# B&R Automation Studio project AAU12Segmenter
Automation Studio 4.12.2.93; technology packages: mapp 5.16.1, mapp6D 1.2.47924, mappCockpit 5.16.0, mappMotion 5.16.2, mappView 5.16.1, mappVision 5.16.1

## Configuration Config1

CPU X20CP1685, AutomationRuntime B4.91, Build 6.3.0, Safety 0.0, Vc V4.72.3

### Task classes (Cpu.sw)
```
Cyclic#1 (cycle 1000 us, tolerance 0 us):
  Main <- Modules.Main.Main.prg
  Acopos6D <- Modules.Acopos6D.Acopos6D.prg
  Vision <- Modules.Services.HMI.Vision.Vision.prg
  Vi_main <- Modules.Services.HMI.Vision.Vi_main.prg
  CTRL <- Modules.KUKA.CTRL.prg
Cyclic#4:
  HMI <- Modules.Services.HMI.HMI.prg
NcDataObjects: mcdrivelog
Binaries: FWRules, arcoal, arsvcreg, TCData, arflatprv, udbdef, mvLoader, mCoWebSc, User, iomap, Config_1, Role, arconfig, asfw, ashwac, sysconf, ashwd, Config_2, viApp, viComp, Settings, Settings_1, asnxdb1
Libraries: standard, brdkMU, brdkSTR, AsSem, sys_lib, brsystem, runtime, AsBrStr, McBase, AsZip, FileIO, AsARCfg, AsEPL, AsIO, astime, ViBase, IecCheck, CoTrace, brdkViBase, brdkViCal, brdkViGeom, brdkViImg, brdkViMapp, brdkViVF, BRSE_RTK, AsHttp, powerlnk, MTLinAlg, McAcp6D, SfDomain, MpBase, KUKAmxA3_1, AsIecCon, MpSfDomMgr, SfDomDrv, SfDomVis, asiodiag, aruser, asusb, arssl, astcp, AsUDP, asstring
```

### Hardware
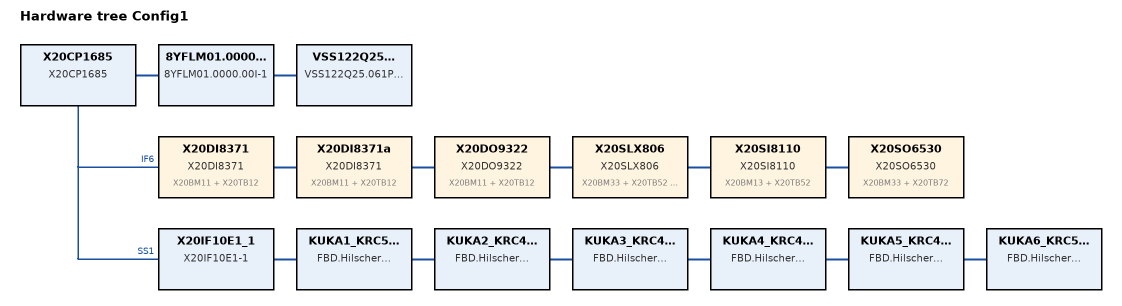
```
8YFLM01.0000.00I-1 : 8YFLM01.0000.00I-1 v0.0.0.1  [PLK1 -> X20CP1685.IF3 (NodeNumber=20) [Cable Type=PowerlinkCable, Length=10, Version=1.0.0.3]; PLK2 -> VSS122Q25.061P-000.PLK1 (NodeNumber=20) [Cable Type=PowerlinkCable, Length=10, Version=1.0.0.3]]
  Supervision = off
KUKA1_KRC5_ProfiNet_6_0 : FBD.Hilscher.PNIOGenDevDTM2.KUKA.PROFINET 6.0 v6.0 (OrderNumber=KUKA.PROFINET 6.0, VendorAddress=krc5-kuka1)  [PN1 -> X20IF10E1_1.IF1]
  DtmId = ed41ecf2-1ee6-4f16-8b0b-5a01acdc12f0
KUKA2_KRC4_ProfiNet_5_0 : FBD.Hilscher.PNIOGenDevDTM2.KRC4-ProfiNet_5.0 v5.0 (OrderNumber=KRC4-ProfiNet_5.0, VendorAddress=krc4-kuka2)  [PN1 -> KUKA1_KRC5_ProfiNet_6_0.PN2]
  DtmId = 37a7288f-95e5-4596-a95a-4f98395b86d6
KUKA3_KRC4_ProfiNet_5_0 : FBD.Hilscher.PNIOGenDevDTM2.KRC4-ProfiNet_5.0 v5.0 (OrderNumber=KRC4-ProfiNet_5.0, VendorAddress=krc4-kuka3)  [PN1 -> KUKA2_KRC4_ProfiNet_5_0.PN2]
  DtmId = 4619762a-1bda-4186-a1d7-16f7a0121dc3
KUKA4_KRC4_ProfiNet_5_0 : FBD.Hilscher.PNIOGenDevDTM2.KRC4-ProfiNet_5.0 v5.0 (OrderNumber=KRC4-ProfiNet_5.0, VendorAddress=krc4-kuka4)  [PN1 -> KUKA3_KRC4_ProfiNet_5_0.PN2]
  DtmId = 587b3b89-59c9-4dff-ae3f-6513934acbe2
KUKA5_KRC4_ProfiNet_5_0 : FBD.Hilscher.PNIOGenDevDTM2.KRC4-ProfiNet_5.0 v5.0 (OrderNumber=KRC4-ProfiNet_5.0, VendorAddress=krc4-kuka5)  [PN1 -> KUKA4_KRC4_ProfiNet_5_0.PN2]
  DtmId = 53f0387d-dc6f-4ff4-995c-9012f8d162e6
KUKA6_KRC5_ProfiNet_6_0 : FBD.Hilscher.PNIOGenDevDTM2.KUKA.PROFINET 6.0 v6.0 (OrderNumber=KUKA.PROFINET 6.0, VendorAddress=krc5-kuka6)  [PN1 -> KUKA5_KRC4_ProfiNet_5_0.PN2]
  DtmId = 2ed1eaca-6452-4986-be94-ac49d0fbd28d
VSS122Q25.061P-000 : VSS122Q25.061P-000 v1.6.0.546  [PLK1 -> 8YFLM01.0000.00I-1.PLK2 (NodeNumber=8) [Cable Type=PowerlinkCable, Length=10, Version=1.0.0.3]]
  Supervision = off
  VisionConfig = gCamera
X20BM11 : X20BM11 v1.1.0.0  [X2X1 -> X20CP1685.IF6]
X20BM11a : X20BM11 v1.1.0.0  [X2X1 -> X20BM11.X2X2]
X20BM11b : X20BM11 v1.1.0.0  [X2X1 -> X20BM11a.X2X2]
X20BM13 : X20BM13 v1.1.0.0  [X2X1 -> X20BM33.X2X2]
X20BM33 : X20BM33 v1.1.0.0  [X2X1 -> X20BM11b.X2X2]
X20BM33a : X20BM33 v1.1.0.0  [X2X1 -> X20BM13.X2X2]
X20CP1685 : X20CP1685 v1.4.0.0
  Connector IF2:
    ActivateDevice = 1
    Mode = Manual
    InternetAddress = 192.168.10.116
    SubnetMask = 255.255.255.0
    ActivateSnmp = 2
  Connector IF3:
    MtuSize = 1500
    DNAConfiguration = manual
    CycleTime = 1000
    InternetAddress = 192.168.200.240
    SubnetMask = 255.255.255.0
  ConfigurationID = Mapp6DDemoKit_Config1
  Simulation = 1
  PermanentPvSize = 6000
  RemanentGlobalPvSize = 40960
  VolatileGlobalPvSize = 200000
  TimerDeviceType = EPLX2X
  TimerDevice = X20CP1685.IF3
  Cyclic1Duration = 1000
  Cyclic1Tolerance = 0
  Cyclic2Duration = 8000
  Cyclic2Tolerance = 16000
  FileDevice1
  FileDeviceName1 = 6DData
  FileDevicePath1 = C:\
  FtpUser1
  FtpUsername1 = admin
  FtpUserPassword1 = jjEtgDO18IYHMAyC5LDIr++62vvoTF/vocBmfWTI62I=  // admin
  FtpUserSalt1 = E9oQkUbZ
  FTPAccessRight1 = 0
  FTPdevice1 = ALL
  ActivateOpcUa = 1
  OpcUaInformationModels_PV_Version = 1
X20DI8371 : X20DI8371 v1.4.0.0  [SS1 -> X20TB12.SS; SL -> X20BM11.SL1]
  Supervision = off
X20DI8371a : X20DI8371 v1.4.0.0  [SS1 -> X20TB12a.SS; SL -> X20BM11a.SL1]
X20DO9322 : X20DO9322 v1.5.0.0  [SS1 -> X20TB12b.SS; SL -> X20BM11b.SL1]
X20IF10E1_1 : X20IF10E1-1 v1.3.0.0  [SS -> X20CP1685.SS1]
  Connector IF1:
    DtmRef = FBDIF.Hilscher.PNIOControllerDTM2.NETX 100 RE/PNM
    DtmId = 9d996fcc-0d20-45c6-b313-689b61703394
  ConfigFile = X20IF10E1_1.dtm
  ConfigModule = asnxdb1
  CycleTime = 1000
X20SI8110 : X20SI8110 v2.4.0.0  [SS1 -> X20TB52b.SS; SL -> X20BM13.SL1]
X20SLX806 : X20SLX806 v2.4.1.1  [SS1 -> X20TB52.SS; SS2 -> X20TB52a.SS; SL -> X20BM33.SL1]
X20SO6530 : X20SO6530 v2.5.0.0  [SS1 -> X20TB72.SS; SL -> X20BM33a.SL1]
  SafeModuleID = 3
X20TB12 : X20TB12 v1.0.0.0
X20TB12a : X20TB12 v1.0.0.0
X20TB12b : X20TB12 v1.0.0.0
X20TB52 : X20TB52 v1.0.0.2
X20TB52a : X20TB52 v1.0.0.2
X20TB52b : X20TB52 v1.0.0.2
X20TB72 : X20TB72 v1.0.0.2
```

### IoMap.iom - X20CP1685/IoMap.iom
```iecst
VAR_CONFIG

	Cyclic#1.::FBin.Array[0] AT %IW."8YFLM01.0000.00I-1".EPL_FB_IN_0_I2007_S01;
	Cyclic#1.::FBin.Array[1] AT %IW."8YFLM01.0000.00I-1".EPL_FB_IN_1_I2007_S02;
	Cyclic#1.::FBin.Array[2] AT %IW."8YFLM01.0000.00I-1".EPL_FB_IN_2_I2007_S03;
	Cyclic#1.::FBin.Array[3] AT %IW."8YFLM01.0000.00I-1".EPL_FB_IN_3_I2007_S04;
	Cyclic#1.::FBin.Array[4] AT %IW."8YFLM01.0000.00I-1".EPL_FB_IN_4_I2007_S05;
	Cyclic#1.::FBin.Array[5] AT %IW."8YFLM01.0000.00I-1".EPL_FB_IN_5_I2007_S06;
	Cyclic#1.::FBin.Array[6] AT %IW."8YFLM01.0000.00I-1".EPL_FB_IN_6_I2007_S07;
	Cyclic#1.::FBin.Array[7] AT %IW."8YFLM01.0000.00I-1".EPL_FB_IN_7_I2007_S08;
	Cyclic#1.::FBin.Array[8] AT %IW."8YFLM01.0000.00I-1".EPL_FB_IN_8_I2007_S09;
	Cyclic#1.::FBin.Array[9] AT %IW."8YFLM01.0000.00I-1".EPL_FB_IN_9_I2007_S0A;
	Cyclic#1.::FBin.Array[10] AT %IW."8YFLM01.0000.00I-1".EPL_FB_IN_10_I2007_S0B;
	Cyclic#1.::FBin.Array[11] AT %IW."8YFLM01.0000.00I-1".EPL_FB_IN_11_I2007_S0C;
	Cyclic#1.::FBin.Array[12] AT %IW."8YFLM01.0000.00I-1".EPL_FB_IN_12_I2007_S0D;
	Cyclic#1.::FBin.Array[13] AT %IW."8YFLM01.0000.00I-1".EPL_FB_IN_13_I2007_S0E;
	Cyclic#1.::FBin.Array[14] AT %IW."8YFLM01.0000.00I-1".EPL_FB_IN_14_I2007_S0F;
	Cyclic#1.::FBin.Array[15] AT %IW."8YFLM01.0000.00I-1".EPL_FB_IN_15_I2007_S10;
	Cyclic#1.::FBin.Array[16] AT %IW."8YFLM01.0000.00I-1".EPL_FB_IN_16_I2007_S11;
	Cyclic#1.::FBin.Array[17] AT %IW."8YFLM01.0000.00I-1".EPL_FB_IN_17_I2007_S12;
	Cyclic#1.::FBin.Array[18] AT %IW."8YFLM01.0000.00I-1".EPL_FB_IN_18_I2007_S13;
	Cyclic#1.::FBin.Array[19] AT %IW."8YFLM01.0000.00I-1".EPL_FB_IN_19_I2007_S14;
	Cyclic#1.::FBin.Array[20] AT %IW."8YFLM01.0000.00I-1".EPL_FB_IN_20_I2007_S15;
	Cyclic#1.::FBin.Array[21] AT %IW."8YFLM01.0000.00I-1".EPL_FB_IN_21_I2007_S16;
	Cyclic#1.::FBin.Array[22] AT %IW."8YFLM01.0000.00I-1".EPL_FB_IN_22_I2007_S17;
	Cyclic#1.::FBin.Array[23] AT %IW."8YFLM01.0000.00I-1".EPL_FB_IN_23_I2007_S18;
	Cyclic#1.::FBin.Array[24] AT %IW."8YFLM01.0000.00I-1".EPL_FB_IN_24_I2007_S19;
	Cyclic#1.::FBin.Array[25] AT %IW."8YFLM01.0000.00I-1".EPL_FB_IN_25_I2007_S1A;
	Cyclic#1.::FBin.Array[26] AT %IW."8YFLM01.0000.00I-1".EPL_FB_IN_26_I2007_S1B;
	Cyclic#1.::FBin.Array[27] AT %IW."8YFLM01.0000.00I-1".EPL_FB_IN_27_I2007_S1C;
	Cyclic#1.::FBin.Array[28] AT %IW."8YFLM01.0000.00I-1".EPL_FB_IN_28_I2007_S1D;
	Cyclic#1.::FBin.Array[29] AT %IW."8YFLM01.0000.00I-1".EPL_FB_IN_29_I2007_S1E;
	Cyclic#1.::FBin.Array[30] AT %IW."8YFLM01.0000.00I-1".EPL_FB_IN_30_I2007_S1F;
	Cyclic#1.::FBin.Array[31] AT %IW."8YFLM01.0000.00I-1".EPL_FB_IN_31_I2007_S20;
	Cyclic#1.::FBin.Array[32] AT %IW."8YFLM01.0000.00I-1".EPL_FB_IN_32_I2007_S21;
	Cyclic#1.::FBin.Array[33] AT %IW."8YFLM01.0000.00I-1".EPL_FB_IN_33_I2007_S22;
	Cyclic#1.::FBin.Array[34] AT %IW."8YFLM01.0000.00I-1".EPL_FB_IN_34_I2007_S23;
	Cyclic#1.::FBin.Array[35] AT %IW."8YFLM01.0000.00I-1".EPL_FB_IN_35_I2007_S24;
	Cyclic#1.::FBin.Array[36] AT %IW."8YFLM01.0000.00I-1".EPL_FB_IN_36_I2007_S25;
	Cyclic#1.::FBin.Array[37] AT %IW."8YFLM01.0000.00I-1".EPL_FB_IN_37_I2007_S26;
	Cyclic#1.::FBin.Array[38] AT %IW."8YFLM01.0000.00I-1".EPL_FB_IN_38_I2007_S27;
	Cyclic#1.::FBin.Array[39] AT %IW."8YFLM01.0000.00I-1".EPL_FB_IN_39_I2007_S28;
	Cyclic#1.::FBin.Array[40] AT %IW."8YFLM01.0000.00I-1".EPL_FB_IN_40_I2007_S29;
	Cyclic#1.::FBin.Array[41] AT %IW."8YFLM01.0000.00I-1".EPL_FB_IN_41_I2007_S2A;
	Cyclic#1.::FBin.Array[42] AT %IW."8YFLM01.0000.00I-1".EPL_FB_IN_42_I2007_S2B;
	Cyclic#1.::FBin.Array[43] AT %IW."8YFLM01.0000.00I-1".EPL_FB_IN_43_I2007_S2C;
	Cyclic#1.::FBin.Array[44] AT %IW."8YFLM01.0000.00I-1".EPL_FB_IN_44_I2007_S2D;
	Cyclic#1.::FBin.Array[45] AT %IW."8YFLM01.0000.00I-1".EPL_FB_IN_45_I2007_S2E;
	Cyclic#1.::FBin.Array[46] AT %IW."8YFLM01.0000.00I-1".EPL_FB_IN_46_I2007_S2F;
	Cyclic#1.::FBin.Array[47] AT %IW."8YFLM01.0000.00I-1".EPL_FB_IN_47_I2007_S30;
	Cyclic#1.::FBin.Array[48] AT %IW."8YFLM01.0000.00I-1".EPL_FB_IN_48_I2007_S31;
	Cyclic#1.::FBin.Array[49] AT %IW."8YFLM01.0000.00I-1".EPL_FB_IN_49_I2007_S32;
	Cyclic#1.::FBin.Array[50] AT %IW."8YFLM01.0000.00I-1".EPL_FB_IN_50_I2007_S33;
	Cyclic#1.::FBin.Array[51] AT %IW."8YFLM01.0000.00I-1".EPL_FB_IN_51_I2007_S34;
	Cyclic#1.::FBin.Array[52] AT %IW."8YFLM01.0000.00I-1".EPL_FB_IN_52_I2007_S35;
	Cyclic#1.::FBin.Array[53] AT %IW."8YFLM01.0000.00I-1".EPL_FB_IN_53_I2007_S36;
	Cyclic#1.::FBin.Array[54] AT %IW."8YFLM01.0000.00I-1".EPL_FB_IN_54_I2007_S37;
	Cyclic#1.::FBin.Array[55] AT %IW."8YFLM01.0000.00I-1".EPL_FB_IN_55_I2007_S38;
	Cyclic#1.::FBin.Array[56] AT %IW."8YFLM01.0000.00I-1".EPL_FB_IN_56_I2007_S39;
	Cyclic#1.::FBin.Array[57] AT %IW."8YFLM01.0000.00I-1".EPL_FB_IN_57_I2007_S3A;
	Cyclic#1.::FBin.Array[58] AT %IW."8YFLM01.0000.00I-1".EPL_FB_IN_58_I2007_S3B;
	Cyclic#1.::FBin.Array[59] AT %IW."8YFLM01.0000.00I-1".EPL_FB_IN_59_I2007_S3C;
	Cyclic#1.::FBin.Array[60] AT %IW."8YFLM01.0000.00I-1".EPL_FB_IN_60_I2007_S3D;
	Cyclic#1.::FBin.Array[61] AT %IW."8YFLM01.0000.00I-1".EPL_FB_IN_61_I2007_S3E;
	Cyclic#1.::FBin.Array[62] AT %IW."8YFLM01.0000.00I-1".EPL_FB_IN_62_I2007_S3F;
	Cyclic#1.::FBin.Array[63] AT %IW."8YFLM01.0000.00I-1".EPL_FB_IN_63_I2007_S40;
	Cyclic#1.::FBin.Array[64] AT %IW."8YFLM01.0000.00I-1".EPL_FB_IN_64_I2007_S41;
	Cyclic#1.::FBin.Array[65] AT %IW."8YFLM01.0000.00I-1".EPL_FB_IN_65_I2007_S42;
	Cyclic#1.::FBin.Array[66] AT %IW."8YFLM01.0000.00I-1".EPL_FB_IN_66_I2007_S43;
	Cyclic#1.::FBin.Array[67] AT %IW."8YFLM01.0000.00I-1".EPL_FB_IN_67_I2007_S44;
	Cyclic#1.::FBin.Array[68] AT %IW."8YFLM01.0000.00I-1".EPL_FB_IN_68_I2007_S45;
	Cyclic#1.::FBin.Array[69] AT %IW."8YFLM01.0000.00I-1".EPL_FB_IN_69_I2007_S46;
	Cyclic#1.::FBin.Array[70] AT %IW."8YFLM01.0000.00I-1".EPL_FB_IN_70_I2007_S47;
	Cyclic#1.::FBin.Array[71] AT %IW."8YFLM01.0000.00I-1".EPL_FB_IN_71_I2007_S48;
	Cyclic#1.::FBin.Array[72] AT %IW."8YFLM01.0000.00I-1".EPL_FB_IN_72_I2007_S49;
	Cyclic#1.::FBin.Array[73] AT %IW."8YFLM01.0000.00I-1".EPL_FB_IN_73_I2007_S4A;
	Cyclic#1.::FBin.Array[74] AT %IW."8YFLM01.0000.00I-1".EPL_FB_IN_74_I2007_S4B;
	Cyclic#1.::FBin.Array[75] AT %IW."8YFLM01.0000.00I-1".EPL_FB_IN_75_I2007_S4C;
	Cyclic#1.::FBin.Array[76] AT %IW."8YFLM01.0000.00I-1".EPL_FB_IN_76_I2007_S4D;
	Cyclic#1.::FBin.Array[77] AT %IW."8YFLM01.0000.00I-1".EPL_FB_IN_77_I2007_S4E;
	Cyclic#1.::FBin.Array[78] AT %IW."8YFLM01.0000.00I-1".EPL_FB_IN_78_I2007_S4F;
	Cyclic#1.::FBin.Array[79] AT %IW."8YFLM01.0000.00I-1".EPL_FB_IN_79_I2007_S50;
	Cyclic#1.::FBin.Array[80] AT %IW."8YFLM01.0000.00I-1".EPL_FB_IN_80_I2007_S51;
	Cyclic#1.::FBin.Array[81] AT %IW."8YFLM01.0000.00I-1".EPL_FB_IN_81_I2007_S52;
	Cyclic#1.::FBin.Array[82] AT %IW."8YFLM01.0000.00I-1".EPL_FB_IN_82_I2007_S53;
	Cyclic#1.::FBin.Array[83] AT %IW."8YFLM01.0000.00I-1".EPL_FB_IN_83_I2007_S54;
	Cyclic#1.::FBin.Array[84] AT %IW."8YFLM01.0000.00I-1".EPL_FB_IN_84_I2007_S55;
	Cyclic#1.::FBin.Array[85] AT %IW."8YFLM01.0000.00I-1".EPL_FB_IN_85_I2007_S56;
	Cyclic#1.::FBin.Array[86] AT %IW."8YFLM01.0000.00I-1".EPL_FB_IN_86_I2007_S57;
	Cyclic#1.::FBin.Array[87] AT %IW."8YFLM01.0000.00I-1".EPL_FB_IN_87_I2007_S58;
	Cyclic#1.::FBin.Array[88] AT %IW."8YFLM01.0000.00I-1".EPL_FB_IN_88_I2007_S59;
	Cyclic#1.::FBin.Array[89] AT %IW."8YFLM01.0000.00I-1".EPL_FB_IN_89_I2007_S5A;
	Cyclic#1.::FBin.Array[90] AT %IW."8YFLM01.0000.00I-1".EPL_FB_IN_90_I2007_S5B;
	Cyclic#1.::FBin.Array[91] AT %IW."8YFLM01.0000.00I-1".EPL_FB_IN_91_I2007_S5C;
	Cyclic#1.::FBin.Array[92] AT %IW."8YFLM01.0000.00I-1".EPL_FB_IN_92_I2007_S5D;
	Cyclic#1.::FBin.Array[93] AT %IW."8YFLM01.0000.00I-1".EPL_FB_IN_93_I2007_S5E;
	Cyclic#1.::FBin.Array[94] AT %IW."8YFLM01.0000.00I-1".EPL_FB_IN_94_I2007_S5F;
	Cyclic#1.::FBin.Array[95] AT %IW."8YFLM01.0000.00I-1".EPL_FB_IN_95_I2007_S60;
	Cyclic#1.::FBin.Array[96] AT %IW."8YFLM01.0000.00I-1".EPL_FB_IN_96_I2007_S61;
	Cyclic#1.::FBin.Array[97] AT %IW."8YFLM01.0000.00I-1".EPL_FB_IN_97_I2007_S62;
	Cyclic#1.::FBin.Array[98] AT %IW."8YFLM01.0000.00I-1".EPL_FB_IN_98_I2007_S63;
	Cyclic#1.::FBin.Array[99] AT %IW."8YFLM01.0000.00I-1".EPL_FB_IN_99_I2007_S64;
	Cyclic#1.::FBin.Array[100] AT %IW."8YFLM01.0000.00I-1".EPL_FB_IN_100_I2007_S65;
	Cyclic#1.::FBin.Array[101] AT %IW."8YFLM01.0000.00I-1".EPL_FB_IN_101_I2007_S66;
	Cyclic#1.::FBin.Array[102] AT %IW."8YFLM01.0000.00I-1".EPL_FB_IN_102_I2007_S67;
	Cyclic#1.::FBin.Array[103] AT %IW."8YFLM01.0000.00I-1".EPL_FB_IN_103_I2007_S68;
	Cyclic#1.::FBin.Array[104] AT %IW."8YFLM01.0000.00I-1".EPL_FB_IN_104_I2007_S69;
	Cyclic#1.::FBin.Array[105] AT %IW."8YFLM01.0000.00I-1".EPL_FB_IN_105_I2007_S6A;
	Cyclic#1.::FBin.Array[106] AT %IW."8YFLM01.0000.00I-1".EPL_FB_IN_106_I2007_S6B;
	Cyclic#1.::FBin.Array[107] AT %IW."8YFLM01.0000.00I-1".EPL_FB_IN_107_I2007_S6C;
	Cyclic#1.::FBin.Array[108] AT %IW."8YFLM01.0000.00I-1".EPL_FB_IN_108_I2007_S6D;
	Cyclic#1.::FBin.Array[109] AT %IW."8YFLM01.0000.00I-1".EPL_FB_IN_109_I2007_S6E;
	Cyclic#1.::FBin.Array[110] AT %IW."8YFLM01.0000.00I-1".EPL_FB_IN_110_I2007_S6F;
	Cyclic#1.::FBin.Array[111] AT %IW."8YFLM01.0000.00I-1".EPL_FB_IN_111_I2007_S70;
	Cyclic#1.::FBin.Array[112] AT %IW."8YFLM01.0000.00I-1".EPL_FB_IN_112_I2007_S71;
	Cyclic#1.::FBin.Array[113] AT %IW."8YFLM01.0000.00I-1".EPL_FB_IN_113_I2007_S72;
	Cyclic#1.::FBin.Array[114] AT %IW."8YFLM01.0000.00I-1".EPL_FB_IN_114_I2007_S73;
	Cyclic#1.::FBin.Array[115] AT %IW."8YFLM01.0000.00I-1".EPL_FB_IN_115_I2007_S74;
	Cyclic#1.::FBin.Array[116] AT %IW."8YFLM01.0000.00I-1".EPL_FB_IN_116_I2007_S75;
	Cyclic#1.::FBin.Array[117] AT %IW."8YFLM01.0000.00I-1".EPL_FB_IN_117_I2007_S76;
	Cyclic#1.::FBin.Array[118] AT %IW."8YFLM01.0000.00I-1".EPL_FB_IN_118_I2007_S77;
	Cyclic#1.::FBin.Array[119] AT %IW."8YFLM01.0000.00I-1".EPL_FB_IN_119_I2007_S78;
	Cyclic#1.::FBin.Array[120] AT %IW."8YFLM01.0000.00I-1".EPL_FB_IN_120_I2007_S79;
	Cyclic#1.::FBin.Array[121] AT %IW."8YFLM01.0000.00I-1".EPL_FB_IN_121_I2007_S7A;
	Cyclic#1.::FBin.Array[122] AT %IW."8YFLM01.0000.00I-1".EPL_FB_IN_122_I2007_S7B;
	Cyclic#1.::FBin.Array[123] AT %IW."8YFLM01.0000.00I-1".EPL_FB_IN_123_I2007_S7C;
	Cyclic#1.::FBin.Array[124] AT %IW."8YFLM01.0000.00I-1".EPL_FB_IN_124_I2007_S7D;
	Cyclic#1.::FBin.Array[125] AT %IW."8YFLM01.0000.00I-1".EPL_FB_IN_125_I2007_S7E;
	Cyclic#1.::FBin.Array[126] AT %IW."8YFLM01.0000.00I-1".EPL_FB_IN_126_I2007_S7F;
	Cyclic#1.::FBin.Array[127] AT %IW."8YFLM01.0000.00I-1".EPL_FB_IN_127_I2007_S80;
	Cyclic#1.::FBin.Array[128] AT %IW."8YFLM01.0000.00I-1".EPL_FB_IN_128_I2007_S81;
	Cyclic#1.::FBin.Array[129] AT %IW."8YFLM01.0000.00I-1".EPL_FB_IN_129_I2007_S82;
	Cyclic#1.::FBin.Array[130] AT %IW."8YFLM01.0000.00I-1".EPL_FB_IN_130_I2007_S83;
	Cyclic#1.::FBin.Array[131] AT %IW."8YFLM01.0000.00I-1".EPL_FB_IN_131_I2007_S84;
	Cyclic#1.::FBin.Array[132] AT %IW."8YFLM01.0000.00I-1".EPL_FB_IN_132_I2007_S85;
	Cyclic#1.::FBin.Array[133] AT %IW."8YFLM01.0000.00I-1".EPL_FB_IN_133_I2007_S86;
	Cyclic#1.::FBin.Array[134] AT %IW."8YFLM01.0000.00I-1".EPL_FB_IN_134_I2007_S87;
	Cyclic#1.::FBin.Array[135] AT %IW."8YFLM01.0000.00I-1".EPL_FB_IN_135_I2007_S88;
	Cyclic#1.::FBin.Array[136] AT %IW."8YFLM01.0000.00I-1".EPL_FB_IN_136_I2007_S89;
	Cyclic#1.::FBin.Array[137] AT %IW."8YFLM01.0000.00I-1".EPL_FB_IN_137_I2007_S8A;
	Cyclic#1.::FBin.Array[138] AT %IW."8YFLM01.0000.00I-1".EPL_FB_IN_138_I2007_S8B;
	Cyclic#1.::FBin.Array[139] AT %IW."8YFLM01.0000.00I-1".EPL_FB_IN_139_I2007_S8C;
	Cyclic#1.::FBin.Array[140] AT %IW."8YFLM01.0000.00I-1".EPL_FB_IN_140_I2007_S8D;
	Cyclic#1.::FBin.Array[141] AT %IW."8YFLM01.0000.00I-1".EPL_FB_IN_141_I2007_S8E;
	Cyclic#1.::FBin.Array[142] AT %IW."8YFLM01.0000.00I-1".EPL_FB_IN_142_I2007_S8F;
	Cyclic#1.::FBin.Array[143] AT %IW."8YFLM01.0000.00I-1".EPL_FB_IN_143_I2007_S90;
	Cyclic#1.::FBin.Array[144] AT %IW."8YFLM01.0000.00I-1".EPL_FB_IN_144_I2007_S91;
	Cyclic#1.::FBin.Array[145] AT %IW."8YFLM01.0000.00I-1".EPL_FB_IN_145_I2007_S92;
	Cyclic#1.::FBin.Array[146] AT %IW."8YFLM01.0000.00I-1".EPL_FB_IN_146_I2007_S93;
	Cyclic#1.::FBin.Array[147] AT %IW."8YFLM01.0000.00I-1".EPL_FB_IN_147_I2007_S94;
	Cyclic#1.::FBin.Array[148] AT %IW."8YFLM01.0000.00I-1".EPL_FB_IN_148_I2007_S95;
	Cyclic#1.::FBin.Array[149] AT %IW."8YFLM01.0000.00I-1".EPL_FB_IN_149_I2007_S96;
	Cyclic#1.::FBin.Array[150] AT %IW."8YFLM01.0000.00I-1".EPL_FB_IN_150_I2007_S97;
	Cyclic#1.::FBin.Array[151] AT %IW."8YFLM01.0000.00I-1".EPL_FB_IN_151_I2007_S98;
	Cyclic#1.::FBin.Array[152] AT %IW."8YFLM01.0000.00I-1".EPL_FB_IN_152_I2007_S99;
	Cyclic#1.::FBin.Array[153] AT %IW."8YFLM01.0000.00I-1".EPL_FB_IN_153_I2007_S9A;
	Cyclic#1.::FBin.Array[154] AT %IW."8YFLM01.0000.00I-1".EPL_FB_IN_154_I2007_S9B;
	Cyclic#1.::FBin.Array[155] AT %IW."8YFLM01.0000.00I-1".EPL_FB_IN_155_I2007_S9C;
	Cyclic#1.::FBin.Array[156] AT %IW."8YFLM01.0000.00I-1".EPL_FB_IN_156_I2007_S9D;
	Cyclic#1.::FBin.Array[157] AT %IW."8YFLM01.0000.00I-1".EPL_FB_IN_157_I2007_S9E;
	Cyclic#1.::FBin.Array[158] AT %IW."8YFLM01.0000.00I-1".EPL_FB_IN_158_I2007_S9F;
	Cyclic#1.::FBin.Array[159] AT %IW."8YFLM01.0000.00I-1".EPL_FB_IN_159_I2007_SA0;
	Cyclic#1.::FBin.Array[160] AT %IW."8YFLM01.0000.00I-1".EPL_FB_IN_160_I2007_SA1;
	Cyclic#1.::FBin.Array[161] AT %IW."8YFLM01.0000.00I-1".EPL_FB_IN_161_I2007_SA2;
	Cyclic#1.::FBin.Array[162] AT %IW."8YFLM01.0000.00I-1".EPL_FB_IN_162_I2007_SA3;
	Cyclic#1.::FBin.Array[163] AT %IW."8YFLM01.0000.00I-1".EPL_FB_IN_163_I2007_SA4;
	Cyclic#1.::FBin.Array[164] AT %IW."8YFLM01.0000.00I-1".EPL_FB_IN_164_I2007_SA5;
	Cyclic#1.::FBin.Array[165] AT %IW."8YFLM01.0000.00I-1".EPL_FB_IN_165_I2007_SA6;
	Cyclic#1.::FBin.Array[166] AT %IW."8YFLM01.0000.00I-1".EPL_FB_IN_166_I2007_SA7;
	Cyclic#1.::FBin.Array[167] AT %IW."8YFLM01.0000.00I-1".EPL_FB_IN_167_I2007_SA8;
	Cyclic#1.::FBin.Array[168] AT %IW."8YFLM01.0000.00I-1".EPL_FB_IN_168_I2007_SA9;
	Cyclic#1.::FBin.Array[169] AT %IW."8YFLM01.0000.00I-1".EPL_FB_IN_169_I2007_SAA;
	Cyclic#1.::FBin.Array[170] AT %IW."8YFLM01.0000.00I-1".EPL_FB_IN_170_I2007_SAB;
	Cyclic#1.::FBin.Array[171] AT %IW."8YFLM01.0000.00I-1".EPL_FB_IN_171_I2007_SAC;
	Cyclic#1.::FBin.Array[172] AT %IW."8YFLM01.0000.00I-1".EPL_FB_IN_172_I2007_SAD;
	Cyclic#1.::FBin.Array[173] AT %IW."8YFLM01.0000.00I-1".EPL_FB_IN_173_I2007_SAE;
	Cyclic#1.::FBin.Array[174] AT %IW."8YFLM01.0000.00I-1".EPL_FB_IN_174_I2007_SAF;
	Cyclic#1.::FBin.Array[175] AT %IW."8YFLM01.0000.00I-1".EPL_FB_IN_175_I2007_SB0;
	Cyclic#1.::FBin.Array[176] AT %IW."8YFLM01.0000.00I-1".EPL_FB_IN_176_I2007_SB1;
	Cyclic#1.::FBin.Array[177] AT %IW."8YFLM01.0000.00I-1".EPL_FB_IN_177_I2007_SB2;
	Cyclic#1.::FBin.Array[178] AT %IW."8YFLM01.0000.00I-1".EPL_FB_IN_178_I2007_SB3;
	Cyclic#1.::FBin.Array[179] AT %IW."8YFLM01.0000.00I-1".EPL_FB_IN_179_I2007_SB4;
	Cyclic#1.::FBin.Array[180] AT %IW."8YFLM01.0000.00I-1".EPL_FB_IN_180_I2007_SB5;
	Cyclic#1.::FBin.Array[181] AT %IW."8YFLM01.0000.00I-1".EPL_FB_IN_181_I2007_SB6;
	Cyclic#1.::FBin.Array[182] AT %IW."8YFLM01.0000.00I-1".EPL_FB_IN_182_I2007_SB7;
	Cyclic#1.::FBin.Array[183] AT %IW."8YFLM01.0000.00I-1".EPL_FB_IN_183_I2007_SB8;
	Cyclic#1.::FBin.Array[184] AT %IW."8YFLM01.0000.00I-1".EPL_FB_IN_184_I2007_SB9;
	Cyclic#1.::FBin.Array[185] AT %IW."8YFLM01.0000.00I-1".EPL_FB_IN_185_I2007_SBA;
	Cyclic#1.::FBin.Array[186] AT %IW."8YFLM01.0000.00I-1".EPL_FB_IN_186_I2007_SBB;
	Cyclic#1.::FBin.Array[187] AT %IW."8YFLM01.0000.00I-1".EPL_FB_IN_187_I2007_SBC;
	Cyclic#1.::FBin.Array[188] AT %IW."8YFLM01.0000.00I-1".EPL_FB_IN_188_I2007_SBD;
	Cyclic#1.::FBin.Array[189] AT %IW."8YFLM01.0000.00I-1".EPL_FB_IN_189_I2007_SBE;
	Cyclic#1.::FBin.Array[190] AT %IW."8YFLM01.0000.00I-1".EPL_FB_IN_190_I2007_SBF;
	Cyclic#1.::FBin.Array[191] AT %IW."8YFLM01.0000.00I-1".EPL_FB_IN_191_I2007_SC0;
	Cyclic#1.::FBin.Array[192] AT %IW."8YFLM01.0000.00I-1".EPL_FB_IN_192_I2007_SC1;
	Cyclic#1.::FBin.Array[193] AT %IW."8YFLM01.0000.00I-1".EPL_FB_IN_193_I2007_SC2;
	Cyclic#1.::FBin.Array[194] AT %IW."8YFLM01.0000.00I-1".EPL_FB_IN_194_I2007_SC3;
	Cyclic#1.::FBin.Array[195] AT %IW."8YFLM01.0000.00I-1".EPL_FB_IN_195_I2007_SC4;
	Cyclic#1.::FBin.Array[196] AT %IW."8YFLM01.0000.00I-1".EPL_FB_IN_196_I2007_SC5;
	Cyclic#1.::FBin.Array[197] AT %IW."8YFLM01.0000.00I-1".EPL_FB_IN_197_I2007_SC6;
	Cyclic#1.::FBin.Array[198] AT %IW."8YFLM01.0000.00I-1".EPL_FB_IN_198_I2007_SC7;
	Cyclic#1.::FBin.Array[199] AT %IW."8YFLM01.0000.00I-1".EPL_FB_IN_199_I2007_SC8;
	Cyclic#1.::FBout.Array[0] AT %QW."8YFLM01.0000.00I-1".EPL_FB_OUT_0_I2008_S01Out;
	Cyclic#1.::FBout.Array[1] AT %QW."8YFLM01.0000.00I-1".EPL_FB_OUT_1_I2008_S02Out;
	Cyclic#1.::FBout.Array[2] AT %QW."8YFLM01.0000.00I-1".EPL_FB_OUT_2_I2008_S03Out;
	Cyclic#1.::FBout.Array[3] AT %QW."8YFLM01.0000.00I-1".EPL_FB_OUT_3_I2008_S04Out;
	Cyclic#1.::FBout.Array[4] AT %QW."8YFLM01.0000.00I-1".EPL_FB_OUT_4_I2008_S05Out;
	Cyclic#1.::FBout.Array[5] AT %QW."8YFLM01.0000.00I-1".EPL_FB_OUT_5_I2008_S06Out;
	Cyclic#1.::FBout.Array[6] AT %QW."8YFLM01.0000.00I-1".EPL_FB_OUT_6_I2008_S07Out;
	Cyclic#1.::FBout.Array[7] AT %QW."8YFLM01.0000.00I-1".EPL_FB_OUT_7_I2008_S08Out;
	Cyclic#1.::FBout.Array[8] AT %QW."8YFLM01.0000.00I-1".EPL_FB_OUT_8_I2008_S09Out;
	Cyclic#1.::FBout.Array[9] AT %QW."8YFLM01.0000.00I-1".EPL_FB_OUT_9_I2008_S0AOut;
	Cyclic#1.::FBout.Array[10] AT %QW."8YFLM01.0000.00I-1".EPL_FB_OUT_10_I2008_S0BOut;
	Cyclic#1.::FBout.Array[11] AT %QW."8YFLM01.0000.00I-1".EPL_FB_OUT_11_I2008_S0COut;
	Cyclic#1.::FBout.Array[12] AT %QW."8YFLM01.0000.00I-1".EPL_FB_OUT_12_I2008_S0DOut;
	Cyclic#1.::FBout.Array[13] AT %QW."8YFLM01.0000.00I-1".EPL_FB_OUT_13_I2008_S0EOut;
	Cyclic#1.::FBout.Array[14] AT %QW."8YFLM01.0000.00I-1".EPL_FB_OUT_14_I2008_S0FOut;
	Cyclic#1.::FBout.Array[15] AT %QW."8YFLM01.0000.00I-1".EPL_FB_OUT_15_I2008_S10Out;
	Cyclic#1.::FBout.Array[16] AT %QW."8YFLM01.0000.00I-1".EPL_FB_OUT_16_I2008_S11Out;
	Cyclic#1.::FBout.Array[17] AT %QW."8YFLM01.0000.00I-1".EPL_FB_OUT_17_I2008_S12Out;
	Cyclic#1.::FBout.Array[18] AT %QW."8YFLM01.0000.00I-1".EPL_FB_OUT_18_I2008_S13Out;
	Cyclic#1.::FBout.Array[19] AT %QW."8YFLM01.0000.00I-1".EPL_FB_OUT_19_I2008_S14Out;
	Cyclic#1.::FBout.Array[20] AT %QW."8YFLM01.0000.00I-1".EPL_FB_OUT_20_I2008_S15Out;
	Cyclic#1.::FBout.Array[21] AT %QW."8YFLM01.0000.00I-1".EPL_FB_OUT_21_I2008_S16Out;
	Cyclic#1.::FBout.Array[22] AT %QW."8YFLM01.0000.00I-1".EPL_FB_OUT_22_I2008_S17Out;
	Cyclic#1.::FBout.Array[23] AT %QW."8YFLM01.0000.00I-1".EPL_FB_OUT_23_I2008_S18Out;
	Cyclic#1.::FBout.Array[24] AT %QW."8YFLM01.0000.00I-1".EPL_FB_OUT_24_I2008_S19Out;
	Cyclic#1.::FBout.Array[25] AT %QW."8YFLM01.0000.00I-1".EPL_FB_OUT_25_I2008_S1AOut;
	Cyclic#1.::FBout.Array[26] AT %QW."8YFLM01.0000.00I-1".EPL_FB_OUT_26_I2008_S1BOut;
	Cyclic#1.::FBout.Array[27] AT %QW."8YFLM01.0000.00I-1".EPL_FB_OUT_27_I2008_S1COut;
	Cyclic#1.::FBout.Array[28] AT %QW."8YFLM01.0000.00I-1".EPL_FB_OUT_28_I2008_S1DOut;
	Cyclic#1.::FBout.Array[29] AT %QW."8YFLM01.0000.00I-1".EPL_FB_OUT_29_I2008_S1EOut;
	Cyclic#1.::FBout.Array[30] AT %QW."8YFLM01.0000.00I-1".EPL_FB_OUT_30_I2008_S1FOut;
	Cyclic#1.::FBout.Array[31] AT %QW."8YFLM01.0000.00I-1".EPL_FB_OUT_31_I2008_S20Out;
	Cyclic#1.::FBout.Array[32] AT %QW."8YFLM01.0000.00I-1".EPL_FB_OUT_32_I2008_S21Out;
	Cyclic#1.::FBout.Array[33] AT %QW."8YFLM01.0000.00I-1".EPL_FB_OUT_33_I2008_S22Out;
	Cyclic#1.::FBout.Array[34] AT %QW."8YFLM01.0000.00I-1".EPL_FB_OUT_34_I2008_S23Out;
	Cyclic#1.::FBout.Array[35] AT %QW."8YFLM01.0000.00I-1".EPL_FB_OUT_35_I2008_S24Out;
	Cyclic#1.::FBout.Array[36] AT %QW."8YFLM01.0000.00I-1".EPL_FB_OUT_36_I2008_S25Out;
	Cyclic#1.::FBout.Array[37] AT %QW."8YFLM01.0000.00I-1".EPL_FB_OUT_37_I2008_S26Out;
	Cyclic#1.::FBout.Array[38] AT %QW."8YFLM01.0000.00I-1".EPL_FB_OUT_38_I2008_S27Out;
	Cyclic#1.::FBout.Array[39] AT %QW."8YFLM01.0000.00I-1".EPL_FB_OUT_39_I2008_S28Out;
	Cyclic#1.::FBout.Array[40] AT %QW."8YFLM01.0000.00I-1".EPL_FB_OUT_40_I2008_S29Out;
	Cyclic#1.::FBout.Array[41] AT %QW."8YFLM01.0000.00I-1".EPL_FB_OUT_41_I2008_S2AOut;
	Cyclic#1.::FBout.Array[42] AT %QW."8YFLM01.0000.00I-1".EPL_FB_OUT_42_I2008_S2BOut;
	Cyclic#1.::FBout.Array[43] AT %QW."8YFLM01.0000.00I-1".EPL_FB_OUT_43_I2008_S2COut;
	Cyclic#1.::FBout.Array[44] AT %QW."8YFLM01.0000.00I-1".EPL_FB_OUT_44_I2008_S2DOut;
	Cyclic#1.::FBout.Array[45] AT %QW."8YFLM01.0000.00I-1".EPL_FB_OUT_45_I2008_S2EOut;
	Cyclic#1.::FBout.Array[46] AT %QW."8YFLM01.0000.00I-1".EPL_FB_OUT_46_I2008_S2FOut;
	Cyclic#1.::FBout.Array[47] AT %QW."8YFLM01.0000.00I-1".EPL_FB_OUT_47_I2008_S30Out;
	Cyclic#1.::FBout.Array[48] AT %QW."8YFLM01.0000.00I-1".EPL_FB_OUT_48_I2008_S31Out;
	Cyclic#1.::FBout.Array[49] AT %QW."8YFLM01.0000.00I-1".EPL_FB_OUT_49_I2008_S32Out;
	Cyclic#1.::FBout.Array[50] AT %QW."8YFLM01.0000.00I-1".EPL_FB_OUT_50_I2008_S33Out;
	Cyclic#1.::FBout.Array[51] AT %QW."8YFLM01.0000.00I-1".EPL_FB_OUT_51_I2008_S34Out;
	Cyclic#1.::FBout.Array[52] AT %QW."8YFLM01.0000.00I-1".EPL_FB_OUT_52_I2008_S35Out;
	Cyclic#1.::FBout.Array[53] AT %QW."8YFLM01.0000.00I-1".EPL_FB_OUT_53_I2008_S36Out;
	Cyclic#1.::FBout.Array[54] AT %QW."8YFLM01.0000.00I-1".EPL_FB_OUT_54_I2008_S37Out;
	Cyclic#1.::FBout.Array[55] AT %QW."8YFLM01.0000.00I-1".EPL_FB_OUT_55_I2008_S38Out;
	Cyclic#1.::FBout.Array[56] AT %QW."8YFLM01.0000.00I-1".EPL_FB_OUT_56_I2008_S39Out;
	Cyclic#1.::FBout.Array[57] AT %QW."8YFLM01.0000.00I-1".EPL_FB_OUT_57_I2008_S3AOut;
	Cyclic#1.::FBout.Array[58] AT %QW."8YFLM01.0000.00I-1".EPL_FB_OUT_58_I2008_S3BOut;
	Cyclic#1.::FBout.Array[59] AT %QW."8YFLM01.0000.00I-1".EPL_FB_OUT_59_I2008_S3COut;
	Cyclic#1.::FBout.Array[60] AT %QW."8YFLM01.0000.00I-1".EPL_FB_OUT_60_I2008_S3DOut;
	Cyclic#1.::FBout.Array[61] AT %QW."8YFLM01.0000.00I-1".EPL_FB_OUT_61_I2008_S3EOut;
	Cyclic#1.::FBout.Array[62] AT %QW."8YFLM01.0000.00I-1".EPL_FB_OUT_62_I2008_S3FOut;
	Cyclic#1.::FBout.Array[63] AT %QW."8YFLM01.0000.00I-1".EPL_FB_OUT_63_I2008_S40Out;
	Cyclic#1.::FBout.Array[64] AT %QW."8YFLM01.0000.00I-1".EPL_FB_OUT_64_I2008_S41Out;
	Cyclic#1.::FBout.Array[65] AT %QW."8YFLM01.0000.00I-1".EPL_FB_OUT_65_I2008_S42Out;
	Cyclic#1.::FBout.Array[66] AT %QW."8YFLM01.0000.00I-1".EPL_FB_OUT_66_I2008_S43Out;
	Cyclic#1.::FBout.Array[67] AT %QW."8YFLM01.0000.00I-1".EPL_FB_OUT_67_I2008_S44Out;
	Cyclic#1.::FBout.Array[68] AT %QW."8YFLM01.0000.00I-1".EPL_FB_OUT_68_I2008_S45Out;
	Cyclic#1.::FBout.Array[69] AT %QW."8YFLM01.0000.00I-1".EPL_FB_OUT_69_I2008_S46Out;
	Cyclic#1.::FBout.Array[70] AT %QW."8YFLM01.0000.00I-1".EPL_FB_OUT_70_I2008_S47Out;
	Cyclic#1.::FBout.Array[71] AT %QW."8YFLM01.0000.00I-1".EPL_FB_OUT_71_I2008_S48Out;
	Cyclic#1.::FBout.Array[72] AT %QW."8YFLM01.0000.00I-1".EPL_FB_OUT_72_I2008_S49Out;
	Cyclic#1.::FBout.Array[73] AT %QW."8YFLM01.0000.00I-1".EPL_FB_OUT_73_I2008_S4AOut;
	Cyclic#1.::FBout.Array[74] AT %QW."8YFLM01.0000.00I-1".EPL_FB_OUT_74_I2008_S4BOut;
	Cyclic#1.::FBout.Array[75] AT %QW."8YFLM01.0000.00I-1".EPL_FB_OUT_75_I2008_S4COut;
	Cyclic#1.::FBout.Array[76] AT %QW."8YFLM01.0000.00I-1".EPL_FB_OUT_76_I2008_S4DOut;
	Cyclic#1.::FBout.Array[77] AT %QW."8YFLM01.0000.00I-1".EPL_FB_OUT_77_I2008_S4EOut;
	Cyclic#1.::FBout.Array[78] AT %QW."8YFLM01.0000.00I-1".EPL_FB_OUT_78_I2008_S4FOut;
	Cyclic#1.::FBout.Array[79] AT %QW."8YFLM01.0000.00I-1".EPL_FB_OUT_79_I2008_S50Out;
	Cyclic#1.::FBout.Array[80] AT %QW."8YFLM01.0000.00I-1".EPL_FB_OUT_80_I2008_S51Out;
	Cyclic#1.::FBout.Array[81] AT %QW."8YFLM01.0000.00I-1".EPL_FB_OUT_81_I2008_S52Out;
	Cyclic#1.::FBout.Array[82] AT %QW."8YFLM01.0000.00I-1".EPL_FB_OUT_82_I2008_S53Out;
	Cyclic#1.::FBout.Array[83] AT %QW."8YFLM01.0000.00I-1".EPL_FB_OUT_83_I2008_S54Out;
	Cyclic#1.::FBout.Array[84] AT %QW."8YFLM01.0000.00I-1".EPL_FB_OUT_84_I2008_S55Out;
	Cyclic#1.::FBout.Array[85] AT %QW."8YFLM01.0000.00I-1".EPL_FB_OUT_85_I2008_S56Out;
	Cyclic#1.::FBout.Array[86] AT %QW."8YFLM01.0000.00I-1".EPL_FB_OUT_86_I2008_S57Out;
	Cyclic#1.::FBout.Array[87] AT %QW."8YFLM01.0000.00I-1".EPL_FB_OUT_87_I2008_S58Out;
	Cyclic#1.::FBout.Array[88] AT %QW."8YFLM01.0000.00I-1".EPL_FB_OUT_88_I2008_S59Out;
	Cyclic#1.::FBout.Array[89] AT %QW."8YFLM01.0000.00I-1".EPL_FB_OUT_89_I2008_S5AOut;
	Cyclic#1.::FBout.Array[90] AT %QW."8YFLM01.0000.00I-1".EPL_FB_OUT_90_I2008_S5BOut;
	Cyclic#1.::FBout.Array[91] AT %QW."8YFLM01.0000.00I-1".EPL_FB_OUT_91_I2008_S5COut;
	Cyclic#1.::FBout.Array[92] AT %QW."8YFLM01.0000.00I-1".EPL_FB_OUT_92_I2008_S5DOut;
	Cyclic#1.::FBout.Array[93] AT %QW."8YFLM01.0000.00I-1".EPL_FB_OUT_93_I2008_S5EOut;
	Cyclic#1.::FBout.Array[94] AT %QW."8YFLM01.0000.00I-1".EPL_FB_OUT_94_I2008_S5FOut;
	Cyclic#1.::FBout.Array[95] AT %QW."8YFLM01.0000.00I-1".EPL_FB_OUT_95_I2008_S60Out;
	Cyclic#1.::FBout.Array[96] AT %QW."8YFLM01.0000.00I-1".EPL_FB_OUT_96_I2008_S61Out;
	Cyclic#1.::FBout.Array[97] AT %QW."8YFLM01.0000.00I-1".EPL_FB_OUT_97_I2008_S62Out;
	Cyclic#1.::FBout.Array[98] AT %QW."8YFLM01.0000.00I-1".EPL_FB_OUT_98_I2008_S63Out;
	Cyclic#1.::FBout.Array[99] AT %QW."8YFLM01.0000.00I-1".EPL_FB_OUT_99_I2008_S64Out;
	Cyclic#1.::FBout.Array[100] AT %QW."8YFLM01.0000.00I-1".EPL_FB_OUT_100_I2008_S65Out;
	Cyclic#1.::FBout.Array[101] AT %QW."8YFLM01.0000.00I-1".EPL_FB_OUT_101_I2008_S66Out;
	Cyclic#1.::FBout.Array[102] AT %QW."8YFLM01.0000.00I-1".EPL_FB_OUT_102_I2008_S67Out;
	Cyclic#1.::FBout.Array[103] AT %QW."8YFLM01.0000.00I-1".EPL_FB_OUT_103_I2008_S68Out;
	Cyclic#1.::FBout.Array[104] AT %QW."8YFLM01.0000.00I-1".EPL_FB_OUT_104_I2008_S69Out;
	Cyclic#1.::FBout.Array[105] AT %QW."8YFLM01.0000.00I-1".EPL_FB_OUT_105_I2008_S6AOut;
	Cyclic#1.::FBout.Array[106] AT %QW."8YFLM01.0000.00I-1".EPL_FB_OUT_106_I2008_S6BOut;
	Cyclic#1.::FBout.Array[107] AT %QW."8YFLM01.0000.00I-1".EPL_FB_OUT_107_I2008_S6COut;
	Cyclic#1.::FBout.Array[108] AT %QW."8YFLM01.0000.00I-1".EPL_FB_OUT_108_I2008_S6DOut;
	Cyclic#1.::FBout.Array[109] AT %QW."8YFLM01.0000.00I-1".EPL_FB_OUT_109_I2008_S6EOut;
	Cyclic#1.::FBout.Array[110] AT %QW."8YFLM01.0000.00I-1".EPL_FB_OUT_110_I2008_S6FOut;
	Cyclic#1.::FBout.Array[111] AT %QW."8YFLM01.0000.00I-1".EPL_FB_OUT_111_I2008_S70Out;
	Cyclic#1.::FBout.Array[112] AT %QW."8YFLM01.0000.00I-1".EPL_FB_OUT_112_I2008_S71Out;
	Cyclic#1.::FBout.Array[113] AT %QW."8YFLM01.0000.00I-1".EPL_FB_OUT_113_I2008_S72Out;
	Cyclic#1.::FBout.Array[114] AT %QW."8YFLM01.0000.00I-1".EPL_FB_OUT_114_I2008_S73Out;
	Cyclic#1.::FBout.Array[115] AT %QW."8YFLM01.0000.00I-1".EPL_FB_OUT_115_I2008_S74Out;
	Cyclic#1.::FBout.Array[116] AT %QW."8YFLM01.0000.00I-1".EPL_FB_OUT_116_I2008_S75Out;
	Cyclic#1.::FBout.Array[117] AT %QW."8YFLM01.0000.00I-1".EPL_FB_OUT_117_I2008_S76Out;
	Cyclic#1.::FBout.Array[118] AT %QW."8YFLM01.0000.00I-1".EPL_FB_OUT_118_I2008_S77Out;
	Cyclic#1.::FBout.Array[119] AT %QW."8YFLM01.0000.00I-1".EPL_FB_OUT_119_I2008_S78Out;
	Cyclic#1.::FBout.Array[120] AT %QW."8YFLM01.0000.00I-1".EPL_FB_OUT_120_I2008_S79Out;
	Cyclic#1.::FBout.Array[121] AT %QW."8YFLM01.0000.00I-1".EPL_FB_OUT_121_I2008_S7AOut;
	Cyclic#1.::FBout.Array[122] AT %QW."8YFLM01.0000.00I-1".EPL_FB_OUT_122_I2008_S7BOut;
	Cyclic#1.::FBout.Array[123] AT %QW."8YFLM01.0000.00I-1".EPL_FB_OUT_123_I2008_S7COut;
	Cyclic#1.::FBout.Array[124] AT %QW."8YFLM01.0000.00I-1".EPL_FB_OUT_124_I2008_S7DOut;
	Cyclic#1.::FBout.Array[125] AT %QW."8YFLM01.0000.00I-1".EPL_FB_OUT_125_I2008_S7EOut;
	Cyclic#1.::FBout.Array[126] AT %QW."8YFLM01.0000.00I-1".EPL_FB_OUT_126_I2008_S7FOut;
	Cyclic#1.::FBout.Array[127] AT %QW."8YFLM01.0000.00I-1".EPL_FB_OUT_127_I2008_S80Out;
	Cyclic#1.::FBout.Array[128] AT %QW."8YFLM01.0000.00I-1".EPL_FB_OUT_128_I2008_S81Out;
	Cyclic#1.::FBout.Array[129] AT %QW."8YFLM01.0000.00I-1".EPL_FB_OUT_129_I2008_S82Out;
	Cyclic#1.::FBout.Array[130] AT %QW."8YFLM01.0000.00I-1".EPL_FB_OUT_130_I2008_S83Out;
	Cyclic#1.::FBout.Array[131] AT %QW."8YFLM01.0000.00I-1".EPL_FB_OUT_131_I2008_S84Out;
	Cyclic#1.::FBout.Array[132] AT %QW."8YFLM01.0000.00I-1".EPL_FB_OUT_132_I2008_S85Out;
	Cyclic#1.::FBout.Array[133] AT %QW."8YFLM01.0000.00I-1".EPL_FB_OUT_133_I2008_S86Out;
	Cyclic#1.::FBout.Array[134] AT %QW."8YFLM01.0000.00I-1".EPL_FB_OUT_134_I2008_S87Out;
	Cyclic#1.::FBout.Array[135] AT %QW."8YFLM01.0000.00I-1".EPL_FB_OUT_135_I2008_S88Out;
	Cyclic#1.::FBout.Array[136] AT %QW."8YFLM01.0000.00I-1".EPL_FB_OUT_136_I2008_S89Out;
	Cyclic#1.::FBout.Array[137] AT %QW."8YFLM01.0000.00I-1".EPL_FB_OUT_137_I2008_S8AOut;
	Cyclic#1.::FBout.Array[138] AT %QW."8YFLM01.0000.00I-1".EPL_FB_OUT_138_I2008_S8BOut;
	Cyclic#1.::FBout.Array[139] AT %QW."8YFLM01.0000.00I-1".EPL_FB_OUT_139_I2008_S8COut;
	Cyclic#1.::FBout.Array[140] AT %QW."8YFLM01.0000.00I-1".EPL_FB_OUT_140_I2008_S8DOut;
	Cyclic#1.::FBout.Array[141] AT %QW."8YFLM01.0000.00I-1".EPL_FB_OUT_141_I2008_S8EOut;
	Cyclic#1.::FBout.Array[142] AT %QW."8YFLM01.0000.00I-1".EPL_FB_OUT_142_I2008_S8FOut;
	Cyclic#1.::FBout.Array[143] AT %QW."8YFLM01.0000.00I-1".EPL_FB_OUT_143_I2008_S90Out;
	Cyclic#1.::FBout.Array[144] AT %QW."8YFLM01.0000.00I-1".EPL_FB_OUT_144_I2008_S91Out;
	Cyclic#1.::FBout.Array[145] AT %QW."8YFLM01.0000.00I-1".EPL_FB_OUT_145_I2008_S92Out;
	Cyclic#1.::FBout.Array[146] AT %QW."8YFLM01.0000.00I-1".EPL_FB_OUT_146_I2008_S93Out;
	Cyclic#1.::FBout.Array[147] AT %QW."8YFLM01.0000.00I-1".EPL_FB_OUT_147_I2008_S94Out;
	Cyclic#1.::FBout.Array[148] AT %QW."8YFLM01.0000.00I-1".EPL_FB_OUT_148_I2008_S95Out;
	Cyclic#1.::FBout.Array[149] AT %QW."8YFLM01.0000.00I-1".EPL_FB_OUT_149_I2008_S96Out;
	Cyclic#1.::FBout.Array[150] AT %QW."8YFLM01.0000.00I-1".EPL_FB_OUT_150_I2008_S97Out;
	Cyclic#1.::FBout.Array[151] AT %QW."8YFLM01.0000.00I-1".EPL_FB_OUT_151_I2008_S98Out;
	Cyclic#1.::FBout.Array[152] AT %QW."8YFLM01.0000.00I-1".EPL_FB_OUT_152_I2008_S99Out;
	Cyclic#1.::FBout.Array[153] AT %QW."8YFLM01.0000.00I-1".EPL_FB_OUT_153_I2008_S9AOut;
	Cyclic#1.::FBout.Array[154] AT %QW."8YFLM01.0000.00I-1".EPL_FB_OUT_154_I2008_S9BOut;
	Cyclic#1.::FBout.Array[155] AT %QW."8YFLM01.0000.00I-1".EPL_FB_OUT_155_I2008_S9COut;
	Cyclic#1.::FBout.Array[156] AT %QW."8YFLM01.0000.00I-1".EPL_FB_OUT_156_I2008_S9DOut;
	Cyclic#1.::FBout.Array[157] AT %QW."8YFLM01.0000.00I-1".EPL_FB_OUT_157_I2008_S9EOut;
	Cyclic#1.::FBout.Array[158] AT %QW."8YFLM01.0000.00I-1".EPL_FB_OUT_158_I2008_S9FOut;
	Cyclic#1.::FBout.Array[159] AT %QW."8YFLM01.0000.00I-1".EPL_FB_OUT_159_I2008_SA0Out;
	Cyclic#1.::FBout.Array[160] AT %QW."8YFLM01.0000.00I-1".EPL_FB_OUT_160_I2008_SA1Out;
	Cyclic#1.::FBout.Array[161] AT %QW."8YFLM01.0000.00I-1".EPL_FB_OUT_161_I2008_SA2Out;
	Cyclic#1.::FBout.Array[162] AT %QW."8YFLM01.0000.00I-1".EPL_FB_OUT_162_I2008_SA3Out;
	Cyclic#1.::FBout.Array[163] AT %QW."8YFLM01.0000.00I-1".EPL_FB_OUT_163_I2008_SA4Out;
	Cyclic#1.::FBout.Array[164] AT %QW."8YFLM01.0000.00I-1".EPL_FB_OUT_164_I2008_SA5Out;
	Cyclic#1.::FBout.Array[165] AT %QW."8YFLM01.0000.00I-1".EPL_FB_OUT_165_I2008_SA6Out;
	Cyclic#1.::FBout.Array[166] AT %QW."8YFLM01.0000.00I-1".EPL_FB_OUT_166_I2008_SA7Out;
	Cyclic#1.::FBout.Array[167] AT %QW."8YFLM01.0000.00I-1".EPL_FB_OUT_167_I2008_SA8Out;
	Cyclic#1.::FBout.Array[168] AT %QW."8YFLM01.0000.00I-1".EPL_FB_OUT_168_I2008_SA9Out;
	Cyclic#1.::FBout.Array[169] AT %QW."8YFLM01.0000.00I-1".EPL_FB_OUT_169_I2008_SAAOut;
	Cyclic#1.::FBout.Array[170] AT %QW."8YFLM01.0000.00I-1".EPL_FB_OUT_170_I2008_SABOut;
	Cyclic#1.::FBout.Array[171] AT %QW."8YFLM01.0000.00I-1".EPL_FB_OUT_171_I2008_SACOut;
	Cyclic#1.::FBout.Array[172] AT %QW."8YFLM01.0000.00I-1".EPL_FB_OUT_172_I2008_SADOut;
	Cyclic#1.::FBout.Array[173] AT %QW."8YFLM01.0000.00I-1".EPL_FB_OUT_173_I2008_SAEOut;
	Cyclic#1.::FBout.Array[174] AT %QW."8YFLM01.0000.00I-1".EPL_FB_OUT_174_I2008_SAFOut;
	Cyclic#1.::FBout.Array[175] AT %QW."8YFLM01.0000.00I-1".EPL_FB_OUT_175_I2008_SB0Out;
	Cyclic#1.::FBout.Array[176] AT %QW."8YFLM01.0000.00I-1".EPL_FB_OUT_176_I2008_SB1Out;
	Cyclic#1.::FBout.Array[177] AT %QW."8YFLM01.0000.00I-1".EPL_FB_OUT_177_I2008_SB2Out;
	Cyclic#1.::FBout.Array[178] AT %QW."8YFLM01.0000.00I-1".EPL_FB_OUT_178_I2008_SB3Out;
	Cyclic#1.::FBout.Array[179] AT %QW."8YFLM01.0000.00I-1".EPL_FB_OUT_179_I2008_SB4Out;
	Cyclic#1.::FBout.Array[180] AT %QW."8YFLM01.0000.00I-1".EPL_FB_OUT_180_I2008_SB5Out;
	Cyclic#1.::FBout.Array[181] AT %QW."8YFLM01.0000.00I-1".EPL_FB_OUT_181_I2008_SB6Out;
	Cyclic#1.::FBout.Array[182] AT %QW."8YFLM01.0000.00I-1".EPL_FB_OUT_182_I2008_SB7Out;
	Cyclic#1.::FBout.Array[183] AT %QW."8YFLM01.0000.00I-1".EPL_FB_OUT_183_I2008_SB8Out;
	Cyclic#1.::FBout.Array[184] AT %QW."8YFLM01.0000.00I-1".EPL_FB_OUT_184_I2008_SB9Out;
	Cyclic#1.::FBout.Array[185] AT %QW."8YFLM01.0000.00I-1".EPL_FB_OUT_185_I2008_SBAOut;
	Cyclic#1.::FBout.Array[186] AT %QW."8YFLM01.0000.00I-1".EPL_FB_OUT_186_I2008_SBBOut;
	Cyclic#1.::FBout.Array[187] AT %QW."8YFLM01.0000.00I-1".EPL_FB_OUT_187_I2008_SBCOut;
	Cyclic#1.::FBout.Array[188] AT %QW."8YFLM01.0000.00I-1".EPL_FB_OUT_188_I2008_SBDOut;
	Cyclic#1.::FBout.Array[189] AT %QW."8YFLM01.0000.00I-1".EPL_FB_OUT_189_I2008_SBEOut;
	Cyclic#1.::FBout.Array[190] AT %QW."8YFLM01.0000.00I-1".EPL_FB_OUT_190_I2008_SBFOut;
	Cyclic#1.::FBout.Array[191] AT %QW."8YFLM01.0000.00I-1".EPL_FB_OUT_191_I2008_SC0Out;
	Cyclic#1.::FBout.Array[192] AT %QW."8YFLM01.0000.00I-1".EPL_FB_OUT_192_I2008_SC1Out;
	Cyclic#1.::FBout.Array[193] AT %QW."8YFLM01.0000.00I-1".EPL_FB_OUT_193_I2008_SC2Out;
	Cyclic#1.::FBout.Array[194] AT %QW."8YFLM01.0000.00I-1".EPL_FB_OUT_194_I2008_SC3Out;
	Cyclic#1.::FBout.Array[195] AT %QW."8YFLM01.0000.00I-1".EPL_FB_OUT_195_I2008_SC4Out;
	Cyclic#1.::FBout.Array[196] AT %QW."8YFLM01.0000.00I-1".EPL_FB_OUT_196_I2008_SC5Out;
	Cyclic#1.::FBout.Array[197] AT %QW."8YFLM01.0000.00I-1".EPL_FB_OUT_197_I2008_SC6Out;
	Cyclic#1.::FBout.Array[198] AT %QW."8YFLM01.0000.00I-1".EPL_FB_OUT_198_I2008_SC7Out;
	Cyclic#1.::FBout.Array[199] AT %QW."8YFLM01.0000.00I-1".EPL_FB_OUT_199_I2008_SC8Out;
	Cyclic#1.::gVisionSensor[3].HW.Connected AT %IX."VSS122Q25.061P-000".ModuleOk;
	Cyclic#1.::gVisionSensor[3].HW.SerialNumber AT %ID."VSS122Q25.061P-000".SerialNumber;
	Cyclic#1.::gVisionSensor[3].HW.ID AT %ID."VSS122Q25.061P-000".ModuleID;
	Cyclic#1.::gVisionSensor[3].HW.Variant AT %ID."VSS122Q25.061P-000".HardwareVariant;
	Cyclic#1.::gVisionSensor[3].HW.Firmware AT %ID."VSS122Q25.061P-000".FirmwareVersion;
	Cyclic#1.::gVisionSensor[3].DAT.Exposure AT %QD."VSS122Q25.061P-000".ExposureTime01;
	Cyclic#1.::gVisionSensor[3].DAT.FlashSegment AT %QB."VSS122Q25.061P-000".FlashSegment01;
	Cyclic#1.::gVisionSensor[3].DAT.AutoSetupExposure AT %ID."VSS122Q25.061P-000".ReadExposureTime;
	Cyclic#1.::gVisionSensor[3].DAT.Status AT %ID."VSS122Q25.061P-000".CameraStatus;
	Cyclic#1.::gVisionSensor[3].DAT.AutoSetupFocus AT %IW."VSS122Q25.061P-000".ReadFocus;
	Cyclic#1.::gVisionSensor[3].DAT.Focus AT %QW."VSS122Q25.061P-000".SetFocus;
	Cyclic#1.::gVisionSensor[3].DAT.Gain AT %QB."VSS122Q25.061P-000".GainLevel;
	Cyclic#1.::gVisionSensor[3].DAT.AutoSetupGain AT %IB."VSS122Q25.061P-000".ReadGainLevel;
	Cyclic#1.::gVisionSensor[3].DAT.AcquisitionFailedCnt AT %IB."VSS122Q25.061P-000".FailedAcquisitionCnt;
	Cyclic#1.::gVisionSensor[3].DAT.AcquisitionCompletedCnt AT %IB."VSS122Q25.061P-000".CompletedAcquisitionCnt;
	Cyclic#1.::gVisionSensor[3].DAT.AcquisitionAcceptedCnt AT %IB."VSS122Q25.061P-000".AcceptedAcquisitionCnt;
	Cyclic#1.::gVisionSensor[3].DAT.NettimeDelay AT %QD."VSS122Q25.061P-000".DelayNettime01;
	Cyclic#1.::gVisionSensor[3].DAT.FlashColor AT %QB."VSS122Q25.061P-000".FlashColor01;
	Cyclic#1.::gVisionSensor[3].CMD.ImageTrigger AT %QX."VSS122Q25.061P-000".ImageAcquisition;
	Cyclic#1.::gVisionSensor[3].DAT.ImageProcessingActive AT %IX."VSS122Q25.061P-000".ImageProcessingActive;
	Cyclic#1.::gVisionSensor[3].CMD.AutoSetupStartStop AT %QX."VSS122Q25.061P-000".SearchAcquisitionSettings;
	Cyclic#1.::gVisionSensor[3].HW.Undervoltage AT %IX."VSS122Q25.061P-000".UndervoltageError;
	Cyclic#1.::gVisionSensor[3].CMD.ImageTriggerReset AT %QX."VSS122Q25.061P-000".ResetAcquisition;
	Cyclic#1.::gVisionSensor[3].HW.Temperature AT %IB."VSS122Q25.061P-000".SensorTemperature;
	Cyclic#1.::gVisionSensor[3].DAT.LightWarningCnt AT %IB."VSS122Q25.061P-000".LightWarningCnt;
	Cyclic#1.::gVisionSensor[3].DAT.LedColor AT %QB."VSS122Q25.061P-000".StatusLED;
	Cyclic#1.::gVisionSensor[3].HW.DigitalInput01 AT %IX."VSS122Q25.061P-000".DigitalInput01;
	Cyclic#1.::gVisionSensor[3].HW.DigitalOutput01 AT %QX."VSS122Q25.061P-000".DigitalOutput01;
	Cyclic#1.::gVisionSensor[3].HW.DigitalOutputStatus01 AT %IX."VSS122Q25.061P-000".DigitalOutputStatus01;
	Cyclic#1.::gVisionSensor[3].HW.Ready AT %IX."VSS122Q25.061P-000".ImageAcquisitionReady;
	Cyclic#1.::gVisionSensor[3].DAT.IRFilter AT %QX."VSS122Q25.061P-000".IRFilter;
	Cyclic#1.::gVisionSensor[3].DAT.ChromaticLock AT %QX."VSS122Q25.061P-000".ChromaticLock;
	Cyclic#1.::gVisionSensor[3].DAT.ProcessingTimeCamera AT %IW."VSS122Q25.061P-000".CameraProcessingTime;
	Cyclic#1.::gVisionSensor[3].DAT.ImageProcessingError AT %IW."VSS122Q25.061P-000".ImageProcessingError;
	Cyclic#1.::gVisionSensor[3].DAT.ImageNettime AT %ID."VSS122Q25.061P-000".ImageNettime;
	::Vision:visionResults AT %IO."VSS122Q25.061P-000".CodeReaderOutput01;
	::Vision:codeReaderVariable1.enable AT %QX."VSS122Q25.061P-000".Enable;
	::Vision:codeReaderVariable1.enableRobustness AT %QX."VSS122Q25.061P-000".EnableRobustness;
	::Vision:codeReaderVariable1.codeType AT %QB."VSS122Q25.061P-000".SymbolType;
	::Vision:codeReaderVariable1.NumberSearch AT %QB."VSS122Q25.061P-000".NumSearchMax;
	::NettimeCurrent_us AT %ID."X20CP1685".SystemTime;
	::Acopos6D:GripperWhitePin AT %QX."X20DO9322".DigitalOutput01;
	::Acopos6D:GripperBlackPin AT %QX."X20DO9322".DigitalOutput02;

	(*________________________________________*)
	(*_____________KUKA1 Mappings_____________*)
	(*________________________________________*)
	::InputVariables[0,0] AT %IB."KUKA1_KRC5_ProfiNet_6_0".Module001_8_digital_inputs_I_00;
	::InputVariables[0,1] AT %IB."KUKA1_KRC5_ProfiNet_6_0".Module001_8_digital_inputs_I_01;
	::InputVariables[0,2] AT %IB."KUKA1_KRC5_ProfiNet_6_0".Module001_8_digital_inputs_I_02;
	::InputVariables[0,3] AT %IB."KUKA1_KRC5_ProfiNet_6_0".Module001_8_digital_inputs_I_03;
	::InputVariables[0,4] AT %IB."KUKA1_KRC5_ProfiNet_6_0".Module001_8_digital_inputs_I_04;
	::InputVariables[0,5] AT %IB."KUKA1_KRC5_ProfiNet_6_0".Module001_8_digital_inputs_I_05;
	::InputVariables[0,6] AT %IB."KUKA1_KRC5_ProfiNet_6_0".Module001_8_digital_inputs_I_06;
	::InputVariables[0,7] AT %IB."KUKA1_KRC5_ProfiNet_6_0".Module001_8_digital_inputs_I_07;
	::InputVariables[0,8] AT %IB."KUKA1_KRC5_ProfiNet_6_0".Module001_8_digital_inputs_I_08;
	::InputVariables[0,9] AT %IB."KUKA1_KRC5_ProfiNet_6_0".Module001_8_digital_inputs_I_09;
	::InputVariables[0,10] AT %IB."KUKA1_KRC5_ProfiNet_6_0".Module001_8_digital_inputs_I_10;
	::InputVariables[0,11] AT %IB."KUKA1_KRC5_ProfiNet_6_0".Module001_8_digital_inputs_I_11;
	::InputVariables[0,12] AT %IB."KUKA1_KRC5_ProfiNet_6_0".Module001_8_digital_inputs_I_12;
	::InputVariables[0,13] AT %IB."KUKA1_KRC5_ProfiNet_6_0".Module001_8_digital_inputs_I_13;
	::InputVariables[0,14] AT %IB."KUKA1_KRC5_ProfiNet_6_0".Module001_8_digital_inputs_I_14;
	::InputVariables[0,15] AT %IB."KUKA1_KRC5_ProfiNet_6_0".Module001_8_digital_inputs_I_15;
	::InputVariables[0,16] AT %IB."KUKA1_KRC5_ProfiNet_6_0".Module001_8_digital_inputs_I_16;
	::InputVariables[0,17] AT %IB."KUKA1_KRC5_ProfiNet_6_0".Module001_8_digital_inputs_I_17;
	::InputVariables[0,18] AT %IB."KUKA1_KRC5_ProfiNet_6_0".Module001_8_digital_inputs_I_18;
	::InputVariables[0,19] AT %IB."KUKA1_KRC5_ProfiNet_6_0".Module001_8_digital_inputs_I_19;
	::InputVariables[0,20] AT %IB."KUKA1_KRC5_ProfiNet_6_0".Module001_8_digital_inputs_I_20;
	::InputVariables[0,21] AT %IB."KUKA1_KRC5_ProfiNet_6_0".Module001_8_digital_inputs_I_21;
	::InputVariables[0,22] AT %IB."KUKA1_KRC5_ProfiNet_6_0".Module001_8_digital_inputs_I_22;
	::InputVariables[0,23] AT %IB."KUKA1_KRC5_ProfiNet_6_0".Module001_8_digital_inputs_I_23;
	::InputVariables[0,24] AT %IB."KUKA1_KRC5_ProfiNet_6_0".Module001_8_digital_inputs_I_24;
	::InputVariables[0,25] AT %IB."KUKA1_KRC5_ProfiNet_6_0".Module001_8_digital_inputs_I_25;
	::InputVariables[0,26] AT %IB."KUKA1_KRC5_ProfiNet_6_0".Module001_8_digital_inputs_I_26;
	::InputVariables[0,27] AT %IB."KUKA1_KRC5_ProfiNet_6_0".Module001_8_digital_inputs_I_27;
	::InputVariables[0,28] AT %IB."KUKA1_KRC5_ProfiNet_6_0".Module001_8_digital_inputs_I_28;
	::InputVariables[0,29] AT %IB."KUKA1_KRC5_ProfiNet_6_0".Module001_8_digital_inputs_I_29;
	::InputVariables[0,30] AT %IB."KUKA1_KRC5_ProfiNet_6_0".Module001_8_digital_inputs_I_30;
	::InputVariables[0,31] AT %IB."KUKA1_KRC5_ProfiNet_6_0".Module001_8_digital_inputs_I_31;
	::InputVariables[0,32] AT %IB."KUKA1_KRC5_ProfiNet_6_0".Module001_8_digital_inputs_I_32;
	::InputVariables[0,33] AT %IB."KUKA1_KRC5_ProfiNet_6_0".Module001_8_digital_inputs_I_33;
	::InputVariables[0,34] AT %IB."KUKA1_KRC5_ProfiNet_6_0".Module001_8_digital_inputs_I_34;
	::InputVariables[0,35] AT %IB."KUKA1_KRC5_ProfiNet_6_0".Module001_8_digital_inputs_I_35;
	::InputVariables[0,36] AT %IB."KUKA1_KRC5_ProfiNet_6_0".Module001_8_digital_inputs_I_36;
	::InputVariables[0,37] AT %IB."KUKA1_KRC5_ProfiNet_6_0".Module001_8_digital_inputs_I_37;
	::InputVariables[0,38] AT %IB."KUKA1_KRC5_ProfiNet_6_0".Module001_8_digital_inputs_I_38;
	::InputVariables[0,39] AT %IB."KUKA1_KRC5_ProfiNet_6_0".Module001_8_digital_inputs_I_39;
	::InputVariables[0,40] AT %IB."KUKA1_KRC5_ProfiNet_6_0".Module001_8_digital_inputs_I_40;
	::InputVariables[0,41] AT %IB."KUKA1_KRC5_ProfiNet_6_0".Module001_8_digital_inputs_I_41;
	::InputVariables[0,42] AT %IB."KUKA1_KRC5_ProfiNet_6_0".Module001_8_digital_inputs_I_42;
	::InputVariables[0,43] AT %IB."KUKA1_KRC5_ProfiNet_6_0".Module001_8_digital_inputs_I_43;
	::InputVariables[0,44] AT %IB."KUKA1_KRC5_ProfiNet_6_0".Module001_8_digital_inputs_I_44;
	::InputVariables[0,45] AT %IB."KUKA1_KRC5_ProfiNet_6_0".Module001_8_digital_inputs_I_45;
	::InputVariables[0,46] AT %IB."KUKA1_KRC5_ProfiNet_6_0".Module001_8_digital_inputs_I_46;
	::InputVariables[0,47] AT %IB."KUKA1_KRC5_ProfiNet_6_0".Module001_8_digital_inputs_I_47;
	::InputVariables[0,48] AT %IB."KUKA1_KRC5_ProfiNet_6_0".Module001_8_digital_inputs_I_48;
	::InputVariables[0,49] AT %IB."KUKA1_KRC5_ProfiNet_6_0".Module001_8_digital_inputs_I_49;
	::InputVariables[0,50] AT %IB."KUKA1_KRC5_ProfiNet_6_0".Module001_8_digital_inputs_I_50;
	::InputVariables[0,51] AT %IB."KUKA1_KRC5_ProfiNet_6_0".Module001_8_digital_inputs_I_51;
	::InputVariables[0,52] AT %IB."KUKA1_KRC5_ProfiNet_6_0".Module001_8_digital_inputs_I_52;
	::InputVariables[0,53] AT %IB."KUKA1_KRC5_ProfiNet_6_0".Module001_8_digital_inputs_I_53;
	::InputVariables[0,54] AT %IB."KUKA1_KRC5_ProfiNet_6_0".Module001_8_digital_inputs_I_54;
	::InputVariables[0,55] AT %IB."KUKA1_KRC5_ProfiNet_6_0".Module001_8_digital_inputs_I_55;
	::InputVariables[0,56] AT %IB."KUKA1_KRC5_ProfiNet_6_0".Module001_8_digital_inputs_I_56;
	::InputVariables[0,57] AT %IB."KUKA1_KRC5_ProfiNet_6_0".Module001_8_digital_inputs_I_57;
	::InputVariables[0,58] AT %IB."KUKA1_KRC5_ProfiNet_6_0".Module001_8_digital_inputs_I_58;
	::InputVariables[0,59] AT %IB."KUKA1_KRC5_ProfiNet_6_0".Module001_8_digital_inputs_I_59;
	::InputVariables[0,60] AT %IB."KUKA1_KRC5_ProfiNet_6_0".Module001_8_digital_inputs_I_60;
	::InputVariables[0,61] AT %IB."KUKA1_KRC5_ProfiNet_6_0".Module001_8_digital_inputs_I_61;
	::InputVariables[0,62] AT %IB."KUKA1_KRC5_ProfiNet_6_0".Module001_8_digital_inputs_I_62;
	::InputVariables[0,63] AT %IB."KUKA1_KRC5_ProfiNet_6_0".Module001_8_digital_inputs_I_63;
	::InputVariables[0,64] AT %IB."KUKA1_KRC5_ProfiNet_6_0".Module001_8_digital_inputs_I_64;
	::InputVariables[0,65] AT %IB."KUKA1_KRC5_ProfiNet_6_0".Module001_8_digital_inputs_I_65;
	::InputVariables[0,66] AT %IB."KUKA1_KRC5_ProfiNet_6_0".Module001_8_digital_inputs_I_66;
	::InputVariables[0,67] AT %IB."KUKA1_KRC5_ProfiNet_6_0".Module001_8_digital_inputs_I_67;
	::InputVariables[0,68] AT %IB."KUKA1_KRC5_ProfiNet_6_0".Module001_8_digital_inputs_I_68;
	::InputVariables[0,69] AT %IB."KUKA1_KRC5_ProfiNet_6_0".Module001_8_digital_inputs_I_69;
	::InputVariables[0,70] AT %IB."KUKA1_KRC5_ProfiNet_6_0".Module001_8_digital_inputs_I_70;
	::InputVariables[0,71] AT %IB."KUKA1_KRC5_ProfiNet_6_0".Module001_8_digital_inputs_I_71;
	::InputVariables[0,72] AT %IB."KUKA1_KRC5_ProfiNet_6_0".Module001_8_digital_inputs_I_72;
	::InputVariables[0,73] AT %IB."KUKA1_KRC5_ProfiNet_6_0".Module001_8_digital_inputs_I_73;
	::InputVariables[0,74] AT %IB."KUKA1_KRC5_ProfiNet_6_0".Module001_8_digital_inputs_I_74;
	::InputVariables[0,75] AT %IB."KUKA1_KRC5_ProfiNet_6_0".Module001_8_digital_inputs_I_75;
	::InputVariables[0,76] AT %IB."KUKA1_KRC5_ProfiNet_6_0".Module001_8_digital_inputs_I_76;
	::InputVariables[0,77] AT %IB."KUKA1_KRC5_ProfiNet_6_0".Module001_8_digital_inputs_I_77;
	::InputVariables[0,78] AT %IB."KUKA1_KRC5_ProfiNet_6_0".Module001_8_digital_inputs_I_78;
	::InputVariables[0,79] AT %IB."KUKA1_KRC5_ProfiNet_6_0".Module001_8_digital_inputs_I_79;
	::InputVariables[0,80] AT %IB."KUKA1_KRC5_ProfiNet_6_0".Module001_8_digital_inputs_I_80;
	::InputVariables[0,81] AT %IB."KUKA1_KRC5_ProfiNet_6_0".Module001_8_digital_inputs_I_81;
	::InputVariables[0,82] AT %IB."KUKA1_KRC5_ProfiNet_6_0".Module001_8_digital_inputs_I_82;
	::InputVariables[0,83] AT %IB."KUKA1_KRC5_ProfiNet_6_0".Module001_8_digital_inputs_I_83;
	::InputVariables[0,84] AT %IB."KUKA1_KRC5_ProfiNet_6_0".Module001_8_digital_inputs_I_84;
	::InputVariables[0,85] AT %IB."KUKA1_KRC5_ProfiNet_6_0".Module001_8_digital_inputs_I_85;
	::InputVariables[0,86] AT %IB."KUKA1_KRC5_ProfiNet_6_0".Module001_8_digital_inputs_I_86;
	::InputVariables[0,87] AT %IB."KUKA1_KRC5_ProfiNet_6_0".Module001_8_digital_inputs_I_87;
	::InputVariables[0,88] AT %IB."KUKA1_KRC5_ProfiNet_6_0".Module001_8_digital_inputs_I_88;
	::InputVariables[0,89] AT %IB."KUKA1_KRC5_ProfiNet_6_0".Module001_8_digital_inputs_I_89;
	::InputVariables[0,90] AT %IB."KUKA1_KRC5_ProfiNet_6_0".Module001_8_digital_inputs_I_90;
	::InputVariables[0,91] AT %IB."KUKA1_KRC5_ProfiNet_6_0".Module001_8_digital_inputs_I_91;
	::InputVariables[0,92] AT %IB."KUKA1_KRC5_ProfiNet_6_0".Module001_8_digital_inputs_I_92;
	::InputVariables[0,93] AT %IB."KUKA1_KRC5_ProfiNet_6_0".Module001_8_digital_inputs_I_93;
	::InputVariables[0,94] AT %IB."KUKA1_KRC5_ProfiNet_6_0".Module001_8_digital_inputs_I_94;
	::InputVariables[0,95] AT %IB."KUKA1_KRC5_ProfiNet_6_0".Module001_8_digital_inputs_I_95;
	::InputVariables[0,96] AT %IB."KUKA1_KRC5_ProfiNet_6_0".Module001_8_digital_inputs_I_96;
	::InputVariables[0,97] AT %IB."KUKA1_KRC5_ProfiNet_6_0".Module001_8_digital_inputs_I_97;
	::InputVariables[0,98] AT %IB."KUKA1_KRC5_ProfiNet_6_0".Module001_8_digital_inputs_I_98;
	::InputVariables[0,99] AT %IB."KUKA1_KRC5_ProfiNet_6_0".Module001_8_digital_inputs_I_99;
	::InputVariables[0,100] AT %IB."KUKA1_KRC5_ProfiNet_6_0".Module001_8_digital_inputs_I_100;
	::InputVariables[0,101] AT %IB."KUKA1_KRC5_ProfiNet_6_0".Module001_8_digital_inputs_I_101;
	::InputVariables[0,102] AT %IB."KUKA1_KRC5_ProfiNet_6_0".Module001_8_digital_inputs_I_102;
	::InputVariables[0,103] AT %IB."KUKA1_KRC5_ProfiNet_6_0".Module001_8_digital_inputs_I_103;
	::InputVariables[0,104] AT %IB."KUKA1_KRC5_ProfiNet_6_0".Module001_8_digital_inputs_I_104;
	::InputVariables[0,105] AT %IB."KUKA1_KRC5_ProfiNet_6_0".Module001_8_digital_inputs_I_105;
	::InputVariables[0,106] AT %IB."KUKA1_KRC5_ProfiNet_6_0".Module001_8_digital_inputs_I_106;
	::InputVariables[0,107] AT %IB."KUKA1_KRC5_ProfiNet_6_0".Module001_8_digital_inputs_I_107;
	::InputVariables[0,108] AT %IB."KUKA1_KRC5_ProfiNet_6_0".Module001_8_digital_inputs_I_108;
	::InputVariables[0,109] AT %IB."KUKA1_KRC5_ProfiNet_6_0".Module001_8_digital_inputs_I_109;
	::InputVariables[0,110] AT %IB."KUKA1_KRC5_ProfiNet_6_0".Module001_8_digital_inputs_I_110;
	::InputVariables[0,111] AT %IB."KUKA1_KRC5_ProfiNet_6_0".Module001_8_digital_inputs_I_111;
	::InputVariables[0,112] AT %IB."KUKA1_KRC5_ProfiNet_6_0".Module001_8_digital_inputs_I_112;
	::InputVariables[0,113] AT %IB."KUKA1_KRC5_ProfiNet_6_0".Module001_8_digital_inputs_I_113;
	::InputVariables[0,114] AT %IB."KUKA1_KRC5_ProfiNet_6_0".Module001_8_digital_inputs_I_114;
	::InputVariables[0,115] AT %IB."KUKA1_KRC5_ProfiNet_6_0".Module001_8_digital_inputs_I_115;
	::InputVariables[0,116] AT %IB."KUKA1_KRC5_ProfiNet_6_0".Module001_8_digital_inputs_I_116;
	::InputVariables[0,117] AT %IB."KUKA1_KRC5_ProfiNet_6_0".Module001_8_digital_inputs_I_117;
	::InputVariables[0,118] AT %IB."KUKA1_KRC5_ProfiNet_6_0".Module001_8_digital_inputs_I_118;
	::InputVariables[0,119] AT %IB."KUKA1_KRC5_ProfiNet_6_0".Module001_8_digital_inputs_I_119;
	::InputVariables[0,120] AT %IB."KUKA1_KRC5_ProfiNet_6_0".Module001_8_digital_inputs_I_120;
	::InputVariables[0,121] AT %IB."KUKA1_KRC5_ProfiNet_6_0".Module001_8_digital_inputs_I_121;
	::InputVariables[0,122] AT %IB."KUKA1_KRC5_ProfiNet_6_0".Module001_8_digital_inputs_I_122;
	::InputVariables[0,123] AT %IB."KUKA1_KRC5_ProfiNet_6_0".Module001_8_digital_inputs_I_123;
	::InputVariables[0,124] AT %IB."KUKA1_KRC5_ProfiNet_6_0".Module001_8_digital_inputs_I_124;
	::InputVariables[0,125] AT %IB."KUKA1_KRC5_ProfiNet_6_0".Module001_8_digital_inputs_I_125;
	::InputVariables[0,126] AT %IB."KUKA1_KRC5_ProfiNet_6_0".Module001_8_digital_inputs_I_126;
	::InputVariables[0,127] AT %IB."KUKA1_KRC5_ProfiNet_6_0".Module001_8_digital_inputs_I_127;
	::InputVariables[0,128] AT %IB."KUKA1_KRC5_ProfiNet_6_0".Module001_8_digital_inputs_I_128;
	::InputVariables[0,129] AT %IB."KUKA1_KRC5_ProfiNet_6_0".Module001_8_digital_inputs_I_129;
	::InputVariables[0,130] AT %IB."KUKA1_KRC5_ProfiNet_6_0".Module001_8_digital_inputs_I_130;
	::InputVariables[0,131] AT %IB."KUKA1_KRC5_ProfiNet_6_0".Module001_8_digital_inputs_I_131;
	::InputVariables[0,132] AT %IB."KUKA1_KRC5_ProfiNet_6_0".Module001_8_digital_inputs_I_132;
	::InputVariables[0,133] AT %IB."KUKA1_KRC5_ProfiNet_6_0".Module001_8_digital_inputs_I_133;
	::InputVariables[0,134] AT %IB."KUKA1_KRC5_ProfiNet_6_0".Module001_8_digital_inputs_I_134;
	::InputVariables[0,135] AT %IB."KUKA1_KRC5_ProfiNet_6_0".Module001_8_digital_inputs_I_135;
	::InputVariables[0,136] AT %IB."KUKA1_KRC5_ProfiNet_6_0".Module001_8_digital_inputs_I_136;
	::InputVariables[0,137] AT %IB."KUKA1_KRC5_ProfiNet_6_0".Module001_8_digital_inputs_I_137;
	::InputVariables[0,138] AT %IB."KUKA1_KRC5_ProfiNet_6_0".Module001_8_digital_inputs_I_138;
	::InputVariables[0,139] AT %IB."KUKA1_KRC5_ProfiNet_6_0".Module001_8_digital_inputs_I_139;
	::InputVariables[0,140] AT %IB."KUKA1_KRC5_ProfiNet_6_0".Module001_8_digital_inputs_I_140;
	::InputVariables[0,141] AT %IB."KUKA1_KRC5_ProfiNet_6_0".Module001_8_digital_inputs_I_141;
	::InputVariables[0,142] AT %IB."KUKA1_KRC5_ProfiNet_6_0".Module001_8_digital_inputs_I_142;
	::InputVariables[0,143] AT %IB."KUKA1_KRC5_ProfiNet_6_0".Module001_8_digital_inputs_I_143;
	::InputVariables[0,144] AT %IB."KUKA1_KRC5_ProfiNet_6_0".Module001_8_digital_inputs_I_144;
	::InputVariables[0,145] AT %IB."KUKA1_KRC5_ProfiNet_6_0".Module001_8_digital_inputs_I_145;
	::InputVariables[0,146] AT %IB."KUKA1_KRC5_ProfiNet_6_0".Module001_8_digital_inputs_I_146;
	::InputVariables[0,147] AT %IB."KUKA1_KRC5_ProfiNet_6_0".Module001_8_digital_inputs_I_147;
	::InputVariables[0,148] AT %IB."KUKA1_KRC5_ProfiNet_6_0".Module001_8_digital_inputs_I_148;
	::InputVariables[0,149] AT %IB."KUKA1_KRC5_ProfiNet_6_0".Module001_8_digital_inputs_I_149;
	::InputVariables[0,150] AT %IB."KUKA1_KRC5_ProfiNet_6_0".Module001_8_digital_inputs_I_150;
	::InputVariables[0,151] AT %IB."KUKA1_KRC5_ProfiNet_6_0".Module001_8_digital_inputs_I_151;
	::InputVariables[0,152] AT %IB."KUKA1_KRC5_ProfiNet_6_0".Module001_8_digital_inputs_I_152;
	::InputVariables[0,153] AT %IB."KUKA1_KRC5_ProfiNet_6_0".Module001_8_digital_inputs_I_153;
	::InputVariables[0,154] AT %IB."KUKA1_KRC5_ProfiNet_6_0".Module001_8_digital_inputs_I_154;
	::InputVariables[0,155] AT %IB."KUKA1_KRC5_ProfiNet_6_0".Module001_8_digital_inputs_I_155;
	::InputVariables[0,156] AT %IB."KUKA1_KRC5_ProfiNet_6_0".Module001_8_digital_inputs_I_156;
	::InputVariables[0,157] AT %IB."KUKA1_KRC5_ProfiNet_6_0".Module001_8_digital_inputs_I_157;
	::InputVariables[0,158] AT %IB."KUKA1_KRC5_ProfiNet_6_0".Module001_8_digital_inputs_I_158;
	::InputVariables[0,159] AT %IB."KUKA1_KRC5_ProfiNet_6_0".Module001_8_digital_inputs_I_159;
	::InputVariables[0,160] AT %IB."KUKA1_KRC5_ProfiNet_6_0".Module001_8_digital_inputs_I_160;
	::InputVariables[0,161] AT %IB."KUKA1_KRC5_ProfiNet_6_0".Module001_8_digital_inputs_I_161;
	::InputVariables[0,162] AT %IB."KUKA1_KRC5_ProfiNet_6_0".Module001_8_digital_inputs_I_162;
	::InputVariables[0,163] AT %IB."KUKA1_KRC5_ProfiNet_6_0".Module001_8_digital_inputs_I_163;
	::InputVariables[0,164] AT %IB."KUKA1_KRC5_ProfiNet_6_0".Module001_8_digital_inputs_I_164;
	::InputVariables[0,165] AT %IB."KUKA1_KRC5_ProfiNet_6_0".Module001_8_digital_inputs_I_165;
	::InputVariables[0,166] AT %IB."KUKA1_KRC5_ProfiNet_6_0".Module001_8_digital_inputs_I_166;
	::InputVariables[0,167] AT %IB."KUKA1_KRC5_ProfiNet_6_0".Module001_8_digital_inputs_I_167;
	::InputVariables[0,168] AT %IB."KUKA1_KRC5_ProfiNet_6_0".Module001_8_digital_inputs_I_168;
	::InputVariables[0,169] AT %IB."KUKA1_KRC5_ProfiNet_6_0".Module001_8_digital_inputs_I_169;
	::InputVariables[0,170] AT %IB."KUKA1_KRC5_ProfiNet_6_0".Module001_8_digital_inputs_I_170;
	::InputVariables[0,171] AT %IB."KUKA1_KRC5_ProfiNet_6_0".Module001_8_digital_inputs_I_171;
	::InputVariables[0,172] AT %IB."KUKA1_KRC5_ProfiNet_6_0".Module001_8_digital_inputs_I_172;
	::InputVariables[0,173] AT %IB."KUKA1_KRC5_ProfiNet_6_0".Module001_8_digital_inputs_I_173;
	::InputVariables[0,174] AT %IB."KUKA1_KRC5_ProfiNet_6_0".Module001_8_digital_inputs_I_174;
	::InputVariables[0,175] AT %IB."KUKA1_KRC5_ProfiNet_6_0".Module001_8_digital_inputs_I_175;
	::InputVariables[0,176] AT %IB."KUKA1_KRC5_ProfiNet_6_0".Module001_8_digital_inputs_I_176;
	::InputVariables[0,177] AT %IB."KUKA1_KRC5_ProfiNet_6_0".Module001_8_digital_inputs_I_177;
	::InputVariables[0,178] AT %IB."KUKA1_KRC5_ProfiNet_6_0".Module001_8_digital_inputs_I_178;
	::InputVariables[0,179] AT %IB."KUKA1_KRC5_ProfiNet_6_0".Module001_8_digital_inputs_I_179;
	::InputVariables[0,180] AT %IB."KUKA1_KRC5_ProfiNet_6_0".Module001_8_digital_inputs_I_180;
	::InputVariables[0,181] AT %IB."KUKA1_KRC5_ProfiNet_6_0".Module001_8_digital_inputs_I_181;
	::InputVariables[0,182] AT %IB."KUKA1_KRC5_ProfiNet_6_0".Module001_8_digital_inputs_I_182;
	::InputVariables[0,183] AT %IB."KUKA1_KRC5_ProfiNet_6_0".Module001_8_digital_inputs_I_183;
	::InputVariables[0,184] AT %IB."KUKA1_KRC5_ProfiNet_6_0".Module001_8_digital_inputs_I_184;
	::InputVariables[0,185] AT %IB."KUKA1_KRC5_ProfiNet_6_0".Module001_8_digital_inputs_I_185;
	::InputVariables[0,186] AT %IB."KUKA1_KRC5_ProfiNet_6_0".Module001_8_digital_inputs_I_186;
	::InputVariables[0,187] AT %IB."KUKA1_KRC5_ProfiNet_6_0".Module001_8_digital_inputs_I_187;
	::InputVariables[0,188] AT %IB."KUKA1_KRC5_ProfiNet_6_0".Module001_8_digital_inputs_I_188;
	::InputVariables[0,189] AT %IB."KUKA1_KRC5_ProfiNet_6_0".Module001_8_digital_inputs_I_189;
	::InputVariables[0,190] AT %IB."KUKA1_KRC5_ProfiNet_6_0".Module001_8_digital_inputs_I_190;
	::InputVariables[0,191] AT %IB."KUKA1_KRC5_ProfiNet_6_0".Module001_8_digital_inputs_I_191;
	::InputVariables[0,192] AT %IB."KUKA1_KRC5_ProfiNet_6_0".Module001_8_digital_inputs_I_192;
	::InputVariables[0,193] AT %IB."KUKA1_KRC5_ProfiNet_6_0".Module001_8_digital_inputs_I_193;
	::InputVariables[0,194] AT %IB."KUKA1_KRC5_ProfiNet_6_0".Module001_8_digital_inputs_I_194;
	::InputVariables[0,195] AT %IB."KUKA1_KRC5_ProfiNet_6_0".Module001_8_digital_inputs_I_195;
	::InputVariables[0,196] AT %IB."KUKA1_KRC5_ProfiNet_6_0".Module001_8_digital_inputs_I_196;
	::InputVariables[0,197] AT %IB."KUKA1_KRC5_ProfiNet_6_0".Module001_8_digital_inputs_I_197;
	::InputVariables[0,198] AT %IB."KUKA1_KRC5_ProfiNet_6_0".Module001_8_digital_inputs_I_198;
	::InputVariables[0,199] AT %IB."KUKA1_KRC5_ProfiNet_6_0".Module001_8_digital_inputs_I_199;
	::InputVariables[0,200] AT %IB."KUKA1_KRC5_ProfiNet_6_0".Module001_8_digital_inputs_I_200;
	::InputVariables[0,201] AT %IB."KUKA1_KRC5_ProfiNet_6_0".Module001_8_digital_inputs_I_201;
	::InputVariables[0,202] AT %IB."KUKA1_KRC5_ProfiNet_6_0".Module001_8_digital_inputs_I_202;
	::InputVariables[0,203] AT %IB."KUKA1_KRC5_ProfiNet_6_0".Module001_8_digital_inputs_I_203;
	::InputVariables[0,204] AT %IB."KUKA1_KRC5_ProfiNet_6_0".Module001_8_digital_inputs_I_204;
	::InputVariables[0,205] AT %IB."KUKA1_KRC5_ProfiNet_6_0".Module001_8_digital_inputs_I_205;
	::InputVariables[0,206] AT %IB."KUKA1_KRC5_ProfiNet_6_0".Module001_8_digital_inputs_I_206;
	::InputVariables[0,207] AT %IB."KUKA1_KRC5_ProfiNet_6_0".Module001_8_digital_inputs_I_207;
	::InputVariables[0,208] AT %IB."KUKA1_KRC5_ProfiNet_6_0".Module001_8_digital_inputs_I_208;
	::InputVariables[0,209] AT %IB."KUKA1_KRC5_ProfiNet_6_0".Module001_8_digital_inputs_I_209;
	::InputVariables[0,210] AT %IB."KUKA1_KRC5_ProfiNet_6_0".Module001_8_digital_inputs_I_210;
	::InputVariables[0,211] AT %IB."KUKA1_KRC5_ProfiNet_6_0".Module001_8_digital_inputs_I_211;
	::InputVariables[0,212] AT %IB."KUKA1_KRC5_ProfiNet_6_0".Module001_8_digital_inputs_I_212;
	::InputVariables[0,213] AT %IB."KUKA1_KRC5_ProfiNet_6_0".Module001_8_digital_inputs_I_213;
	::InputVariables[0,214] AT %IB."KUKA1_KRC5_ProfiNet_6_0".Module001_8_digital_inputs_I_214;
	::InputVariables[0,215] AT %IB."KUKA1_KRC5_ProfiNet_6_0".Module001_8_digital_inputs_I_215;
	::InputVariables[0,216] AT %IB."KUKA1_KRC5_ProfiNet_6_0".Module001_8_digital_inputs_I_216;
	::InputVariables[0,217] AT %IB."KUKA1_KRC5_ProfiNet_6_0".Module001_8_digital_inputs_I_217;
	::InputVariables[0,218] AT %IB."KUKA1_KRC5_ProfiNet_6_0".Module001_8_digital_inputs_I_218;
	::InputVariables[0,219] AT %IB."KUKA1_KRC5_ProfiNet_6_0".Module001_8_digital_inputs_I_219;
	::InputVariables[0,220] AT %IB."KUKA1_KRC5_ProfiNet_6_0".Module001_8_digital_inputs_I_220;
	::InputVariables[0,221] AT %IB."KUKA1_KRC5_ProfiNet_6_0".Module001_8_digital_inputs_I_221;
	::InputVariables[0,222] AT %IB."KUKA1_KRC5_ProfiNet_6_0".Module001_8_digital_inputs_I_222;
	::InputVariables[0,223] AT %IB."KUKA1_KRC5_ProfiNet_6_0".Module001_8_digital_inputs_I_223;
	::InputVariables[0,224] AT %IB."KUKA1_KRC5_ProfiNet_6_0".Module001_8_digital_inputs_I_224;
	::InputVariables[0,225] AT %IB."KUKA1_KRC5_ProfiNet_6_0".Module001_8_digital_inputs_I_225;
	::InputVariables[0,226] AT %IB."KUKA1_KRC5_ProfiNet_6_0".Module001_8_digital_inputs_I_226;
	::InputVariables[0,227] AT %IB."KUKA1_KRC5_ProfiNet_6_0".Module001_8_digital_inputs_I_227;
	::InputVariables[0,228] AT %IB."KUKA1_KRC5_ProfiNet_6_0".Module001_8_digital_inputs_I_228;
	::InputVariables[0,229] AT %IB."KUKA1_KRC5_ProfiNet_6_0".Module001_8_digital_inputs_I_229;
	::InputVariables[0,230] AT %IB."KUKA1_KRC5_ProfiNet_6_0".Module001_8_digital_inputs_I_230;
	::InputVariables[0,231] AT %IB."KUKA1_KRC5_ProfiNet_6_0".Module001_8_digital_inputs_I_231;
	::InputVariables[0,232] AT %IB."KUKA1_KRC5_ProfiNet_6_0".Module001_8_digital_inputs_I_232;
	::InputVariables[0,233] AT %IB."KUKA1_KRC5_ProfiNet_6_0".Module001_8_digital_inputs_I_233;
	::InputVariables[0,234] AT %IB."KUKA1_KRC5_ProfiNet_6_0".Module001_8_digital_inputs_I_234;
	::InputVariables[0,235] AT %IB."KUKA1_KRC5_ProfiNet_6_0".Module001_8_digital_inputs_I_235;
	::InputVariables[0,236] AT %IB."KUKA1_KRC5_ProfiNet_6_0".Module001_8_digital_inputs_I_236;
	::InputVariables[0,237] AT %IB."KUKA1_KRC5_ProfiNet_6_0".Module001_8_digital_inputs_I_237;
	::InputVariables[0,238] AT %IB."KUKA1_KRC5_ProfiNet_6_0".Module001_8_digital_inputs_I_238;
	::InputVariables[0,239] AT %IB."KUKA1_KRC5_ProfiNet_6_0".Module001_8_digital_inputs_I_239;
	::InputVariables[0,240] AT %IB."KUKA1_KRC5_ProfiNet_6_0".Module001_8_digital_inputs_I_240;
	::InputVariables[0,241] AT %IB."KUKA1_KRC5_ProfiNet_6_0".Module001_8_digital_inputs_I_241;
	::InputVariables[0,242] AT %IB."KUKA1_KRC5_ProfiNet_6_0".Module001_8_digital_inputs_I_242;
	::InputVariables[0,243] AT %IB."KUKA1_KRC5_ProfiNet_6_0".Module001_8_digital_inputs_I_243;
	::InputVariables[0,244] AT %IB."KUKA1_KRC5_ProfiNet_6_0".Module001_8_digital_inputs_I_244;
	::InputVariables[0,245] AT %IB."KUKA1_KRC5_ProfiNet_6_0".Module001_8_digital_inputs_I_245;
	::InputVariables[0,246] AT %IB."KUKA1_KRC5_ProfiNet_6_0".Module001_8_digital_inputs_I_246;
	::InputVariables[0,247] AT %IB."KUKA1_KRC5_ProfiNet_6_0".Module001_8_digital_inputs_I_247;
	::InputVariables[0,248] AT %IB."KUKA1_KRC5_ProfiNet_6_0".Module001_8_digital_inputs_I_248;
	::InputVariables[0,249] AT %IB."KUKA1_KRC5_ProfiNet_6_0".Module001_8_digital_inputs_I_249;
	::InputVariables[0,250] AT %IB."KUKA1_KRC5_ProfiNet_6_0".Module001_8_digital_inputs_I_250;
	::InputVariables[0,251] AT %IB."KUKA1_KRC5_ProfiNet_6_0".Module001_8_digital_inputs_I_251;
	::InputVariables[0,252] AT %IB."KUKA1_KRC5_ProfiNet_6_0".Module001_8_digital_inputs_I_252;
	::InputVariables[0,253] AT %IB."KUKA1_KRC5_ProfiNet_6_0".Module001_8_digital_inputs_I_253;

	::OutputVariables[0,0]	AT %QB."KUKA1_KRC5_ProfiNet_6_0".Module001_8_digital_outputs_O_00;
	::OutputVariables[0,1]	AT %QB."KUKA1_KRC5_ProfiNet_6_0".Module001_8_digital_outputs_O_01;
	::OutputVariables[0,2]	AT %QB."KUKA1_KRC5_ProfiNet_6_0".Module001_8_digital_outputs_O_02;
	::OutputVariables[0,3]	AT %QB."KUKA1_KRC5_ProfiNet_6_0".Module001_8_digital_outputs_O_03;
	::OutputVariables[0,4]	AT %QB."KUKA1_KRC5_ProfiNet_6_0".Module001_8_digital_outputs_O_04;
	::OutputVariables[0,5]	AT %QB."KUKA1_KRC5_ProfiNet_6_0".Module001_8_digital_outputs_O_05;
	::OutputVariables[0,6]	AT %QB."KUKA1_KRC5_ProfiNet_6_0".Module001_8_digital_outputs_O_06;
	::OutputVariables[0,7]	AT %QB."KUKA1_KRC5_ProfiNet_6_0".Module001_8_digital_outputs_O_07;
	::OutputVariables[0,8]	AT %QB."KUKA1_KRC5_ProfiNet_6_0".Module001_8_digital_outputs_O_08;
	::OutputVariables[0,9]	AT %QB."KUKA1_KRC5_ProfiNet_6_0".Module001_8_digital_outputs_O_09;
	::OutputVariables[0,10]	AT %QB."KUKA1_KRC5_ProfiNet_6_0".Module001_8_digital_outputs_O_10;
	::OutputVariables[0,11]	AT %QB."KUKA1_KRC5_ProfiNet_6_0".Module001_8_digital_outputs_O_11;
	::OutputVariables[0,12]	AT %QB."KUKA1_KRC5_ProfiNet_6_0".Module001_8_digital_outputs_O_12;
	::OutputVariables[0,13]	AT %QB."KUKA1_KRC5_ProfiNet_6_0".Module001_8_digital_outputs_O_13;
	::OutputVariables[0,14]	AT %QB."KUKA1_KRC5_ProfiNet_6_0".Module001_8_digital_outputs_O_14;
	::OutputVariables[0,15]	AT %QB."KUKA1_KRC5_ProfiNet_6_0".Module001_8_digital_outputs_O_15;
	::OutputVariables[0,16]	AT %QB."KUKA1_KRC5_ProfiNet_6_0".Module001_8_digital_outputs_O_16;
	::OutputVariables[0,17]	AT %QB."KUKA1_KRC5_ProfiNet_6_0".Module001_8_digital_outputs_O_17;
	::OutputVariables[0,18]	AT %QB."KUKA1_KRC5_ProfiNet_6_0".Module001_8_digital_outputs_O_18;
	::OutputVariables[0,19]	AT %QB."KUKA1_KRC5_ProfiNet_6_0".Module001_8_digital_outputs_O_19;
	::OutputVariables[0,20]	AT %QB."KUKA1_KRC5_ProfiNet_6_0".Module001_8_digital_outputs_O_20;
	::OutputVariables[0,21]	AT %QB."KUKA1_KRC5_ProfiNet_6_0".Module001_8_digital_outputs_O_21;
	::OutputVariables[0,22]	AT %QB."KUKA1_KRC5_ProfiNet_6_0".Module001_8_digital_outputs_O_22;
	::OutputVariables[0,23]	AT %QB."KUKA1_KRC5_ProfiNet_6_0".Module001_8_digital_outputs_O_23;
	::OutputVariables[0,24]	AT %QB."KUKA1_KRC5_ProfiNet_6_0".Module001_8_digital_outputs_O_24;
	::OutputVariables[0,25]	AT %QB."KUKA1_KRC5_ProfiNet_6_0".Module001_8_digital_outputs_O_25;
	::OutputVariables[0,26]	AT %QB."KUKA1_KRC5_ProfiNet_6_0".Module001_8_digital_outputs_O_26;
	::OutputVariables[0,27]	AT %QB."KUKA1_KRC5_ProfiNet_6_0".Module001_8_digital_outputs_O_27;
	::OutputVariables[0,28]	AT %QB."KUKA1_KRC5_ProfiNet_6_0".Module001_8_digital_outputs_O_28;
	::OutputVariables[0,29]	AT %QB."KUKA1_KRC5_ProfiNet_6_0".Module001_8_digital_outputs_O_29;
	::OutputVariables[0,30]	AT %QB."KUKA1_KRC5_ProfiNet_6_0".Module001_8_digital_outputs_O_30;
	::OutputVariables[0,31]	AT %QB."KUKA1_KRC5_ProfiNet_6_0".Module001_8_digital_outputs_O_31;
	::OutputVariables[0,32]	AT %QB."KUKA1_KRC5_ProfiNet_6_0".Module001_8_digital_outputs_O_32;
	::OutputVariables[0,33]	AT %QB."KUKA1_KRC5_ProfiNet_6_0".Module001_8_digital_outputs_O_33;
	::OutputVariables[0,34]	AT %QB."KUKA1_KRC5_ProfiNet_6_0".Module001_8_digital_outputs_O_34;
	::OutputVariables[0,35]	AT %QB."KUKA1_KRC5_ProfiNet_6_0".Module001_8_digital_outputs_O_35;
	::OutputVariables[0,36]	AT %QB."KUKA1_KRC5_ProfiNet_6_0".Module001_8_digital_outputs_O_36;
	::OutputVariables[0,37]	AT %QB."KUKA1_KRC5_ProfiNet_6_0".Module001_8_digital_outputs_O_37;
	::OutputVariables[0,38]	AT %QB."KUKA1_KRC5_ProfiNet_6_0".Module001_8_digital_outputs_O_38;
	::OutputVariables[0,39]	AT %QB."KUKA1_KRC5_ProfiNet_6_0".Module001_8_digital_outputs_O_39;
	::OutputVariables[0,40]	AT %QB."KUKA1_KRC5_ProfiNet_6_0".Module001_8_digital_outputs_O_40;
	::OutputVariables[0,41]	AT %QB."KUKA1_KRC5_ProfiNet_6_0".Module001_8_digital_outputs_O_41;
	::OutputVariables[0,42]	AT %QB."KUKA1_KRC5_ProfiNet_6_0".Module001_8_digital_outputs_O_42;
	::OutputVariables[0,43]	AT %QB."KUKA1_KRC5_ProfiNet_6_0".Module001_8_digital_outputs_O_43;
	::OutputVariables[0,44]	AT %QB."KUKA1_KRC5_ProfiNet_6_0".Module001_8_digital_outputs_O_44;
	::OutputVariables[0,45]	AT %QB."KUKA1_KRC5_ProfiNet_6_0".Module001_8_digital_outputs_O_45;
	::OutputVariables[0,46]	AT %QB."KUKA1_KRC5_ProfiNet_6_0".Module001_8_digital_outputs_O_46;
	::OutputVariables[0,47]	AT %QB."KUKA1_KRC5_ProfiNet_6_0".Module001_8_digital_outputs_O_47;
	::OutputVariables[0,48]	AT %QB."KUKA1_KRC5_ProfiNet_6_0".Module001_8_digital_outputs_O_48;
	::OutputVariables[0,49]	AT %QB."KUKA1_KRC5_ProfiNet_6_0".Module001_8_digital_outputs_O_49;
	::OutputVariables[0,50]	AT %QB."KUKA1_KRC5_ProfiNet_6_0".Module001_8_digital_outputs_O_50;
	::OutputVariables[0,51]	AT %QB."KUKA1_KRC5_ProfiNet_6_0".Module001_8_digital_outputs_O_51;
	::OutputVariables[0,52]	AT %QB."KUKA1_KRC5_ProfiNet_6_0".Module001_8_digital_outputs_O_52;
	::OutputVariables[0,53]	AT %QB."KUKA1_KRC5_ProfiNet_6_0".Module001_8_digital_outputs_O_53;
	::OutputVariables[0,54]	AT %QB."KUKA1_KRC5_ProfiNet_6_0".Module001_8_digital_outputs_O_54;
	::OutputVariables[0,55]	AT %QB."KUKA1_KRC5_ProfiNet_6_0".Module001_8_digital_outputs_O_55;
	::OutputVariables[0,56]	AT %QB."KUKA1_KRC5_ProfiNet_6_0".Module001_8_digital_outputs_O_56;
	::OutputVariables[0,57]	AT %QB."KUKA1_KRC5_ProfiNet_6_0".Module001_8_digital_outputs_O_57;
	::OutputVariables[0,58]	AT %QB."KUKA1_KRC5_ProfiNet_6_0".Module001_8_digital_outputs_O_58;
	::OutputVariables[0,59]	AT %QB."KUKA1_KRC5_ProfiNet_6_0".Module001_8_digital_outputs_O_59;
	::OutputVariables[0,60]	AT %QB."KUKA1_KRC5_ProfiNet_6_0".Module001_8_digital_outputs_O_60;
	::OutputVariables[0,61]	AT %QB."KUKA1_KRC5_ProfiNet_6_0".Module001_8_digital_outputs_O_61;
	::OutputVariables[0,62]	AT %QB."KUKA1_KRC5_ProfiNet_6_0".Module001_8_digital_outputs_O_62;
	::OutputVariables[0,63]	AT %QB."KUKA1_KRC5_ProfiNet_6_0".Module001_8_digital_outputs_O_63;
	::OutputVariables[0,64]	AT %QB."KUKA1_KRC5_ProfiNet_6_0".Module001_8_digital_outputs_O_64;
	::OutputVariables[0,65]	AT %QB."KUKA1_KRC5_ProfiNet_6_0".Module001_8_digital_outputs_O_65;
	::OutputVariables[0,66]	AT %QB."KUKA1_KRC5_ProfiNet_6_0".Module001_8_digital_outputs_O_66;
	::OutputVariables[0,67]	AT %QB."KUKA1_KRC5_ProfiNet_6_0".Module001_8_digital_outputs_O_67;
	::OutputVariables[0,68]	AT %QB."KUKA1_KRC5_ProfiNet_6_0".Module001_8_digital_outputs_O_68;
	::OutputVariables[0,69]	AT %QB."KUKA1_KRC5_ProfiNet_6_0".Module001_8_digital_outputs_O_69;
	::OutputVariables[0,70]	AT %QB."KUKA1_KRC5_ProfiNet_6_0".Module001_8_digital_outputs_O_70;
	::OutputVariables[0,71]	AT %QB."KUKA1_KRC5_ProfiNet_6_0".Module001_8_digital_outputs_O_71;
	::OutputVariables[0,72]	AT %QB."KUKA1_KRC5_ProfiNet_6_0".Module001_8_digital_outputs_O_72;
	::OutputVariables[0,73]	AT %QB."KUKA1_KRC5_ProfiNet_6_0".Module001_8_digital_outputs_O_73;
	::OutputVariables[0,74]	AT %QB."KUKA1_KRC5_ProfiNet_6_0".Module001_8_digital_outputs_O_74;
	::OutputVariables[0,75]	AT %QB."KUKA1_KRC5_ProfiNet_6_0".Module001_8_digital_outputs_O_75;
	::OutputVariables[0,76]	AT %QB."KUKA1_KRC5_ProfiNet_6_0".Module001_8_digital_outputs_O_76;
	::OutputVariables[0,77]	AT %QB."KUKA1_KRC5_ProfiNet_6_0".Module001_8_digital_outputs_O_77;
	::OutputVariables[0,78]	AT %QB."KUKA1_KRC5_ProfiNet_6_0".Module001_8_digital_outputs_O_78;
	::OutputVariables[0,79]	AT %QB."KUKA1_KRC5_ProfiNet_6_0".Module001_8_digital_outputs_O_79;
	::OutputVariables[0,80]	AT %QB."KUKA1_KRC5_ProfiNet_6_0".Module001_8_digital_outputs_O_80;
	::OutputVariables[0,81]	AT %QB."KUKA1_KRC5_ProfiNet_6_0".Module001_8_digital_outputs_O_81;
	::OutputVariables[0,82]	AT %QB."KUKA1_KRC5_ProfiNet_6_0".Module001_8_digital_outputs_O_82;
	::OutputVariables[0,83]	AT %QB."KUKA1_KRC5_ProfiNet_6_0".Module001_8_digital_outputs_O_83;
	::OutputVariables[0,84]	AT %QB."KUKA1_KRC5_ProfiNet_6_0".Module001_8_digital_outputs_O_84;
	::OutputVariables[0,85]	AT %QB."KUKA1_KRC5_ProfiNet_6_0".Module001_8_digital_outputs_O_85;
	::OutputVariables[0,86]	AT %QB."KUKA1_KRC5_ProfiNet_6_0".Module001_8_digital_outputs_O_86;
	::OutputVariables[0,87]	AT %QB."KUKA1_KRC5_ProfiNet_6_0".Module001_8_digital_outputs_O_87;
	::OutputVariables[0,88]	AT %QB."KUKA1_KRC5_ProfiNet_6_0".Module001_8_digital_outputs_O_88;
	::OutputVariables[0,89]	AT %QB."KUKA1_KRC5_ProfiNet_6_0".Module001_8_digital_outputs_O_89;
	::OutputVariables[0,90]	AT %QB."KUKA1_KRC5_ProfiNet_6_0".Module001_8_digital_outputs_O_90;
	::OutputVariables[0,91]	AT %QB."KUKA1_KRC5_ProfiNet_6_0".Module001_8_digital_outputs_O_91;
	::OutputVariables[0,92]	AT %QB."KUKA1_KRC5_ProfiNet_6_0".Module001_8_digital_outputs_O_92;
	::OutputVariables[0,93]	AT %QB."KUKA1_KRC5_ProfiNet_6_0".Module001_8_digital_outputs_O_93;
	::OutputVariables[0,94]	AT %QB."KUKA1_KRC5_ProfiNet_6_0".Module001_8_digital_outputs_O_94;
	::OutputVariables[0,95]	AT %QB."KUKA1_KRC5_ProfiNet_6_0".Module001_8_digital_outputs_O_95;
	::OutputVariables[0,96]	AT %QB."KUKA1_KRC5_ProfiNet_6_0".Module001_8_digital_outputs_O_96;
	::OutputVariables[0,97]	AT %QB."KUKA1_KRC5_ProfiNet_6_0".Module001_8_digital_outputs_O_97;
	::OutputVariables[0,98]	AT %QB."KUKA1_KRC5_ProfiNet_6_0".Module001_8_digital_outputs_O_98;
	::OutputVariables[0,99]	AT %QB."KUKA1_KRC5_ProfiNet_6_0".Module001_8_digital_outputs_O_99;
	::OutputVariables[0,100]	AT %QB."KUKA1_KRC5_ProfiNet_6_0".Module001_8_digital_outputs_O_100;
	::OutputVariables[0,101]	AT %QB."KUKA1_KRC5_ProfiNet_6_0".Module001_8_digital_outputs_O_101;
	::OutputVariables[0,102]	AT %QB."KUKA1_KRC5_ProfiNet_6_0".Module001_8_digital_outputs_O_102;
	::OutputVariables[0,103]	AT %QB."KUKA1_KRC5_ProfiNet_6_0".Module001_8_digital_outputs_O_103;
	::OutputVariables[0,104]	AT %QB."KUKA1_KRC5_ProfiNet_6_0".Module001_8_digital_outputs_O_104;
	::OutputVariables[0,105]	AT %QB."KUKA1_KRC5_ProfiNet_6_0".Module001_8_digital_outputs_O_105;
	::OutputVariables[0,106]	AT %QB."KUKA1_KRC5_ProfiNet_6_0".Module001_8_digital_outputs_O_106;
	::OutputVariables[0,107]	AT %QB."KUKA1_KRC5_ProfiNet_6_0".Module001_8_digital_outputs_O_107;
	::OutputVariables[0,108]	AT %QB."KUKA1_KRC5_ProfiNet_6_0".Module001_8_digital_outputs_O_108;
	::OutputVariables[0,109]	AT %QB."KUKA1_KRC5_ProfiNet_6_0".Module001_8_digital_outputs_O_109;
	::OutputVariables[0,110]	AT %QB."KUKA1_KRC5_ProfiNet_6_0".Module001_8_digital_outputs_O_110;
	::OutputVariables[0,111]	AT %QB."KUKA1_KRC5_ProfiNet_6_0".Module001_8_digital_outputs_O_111;
	::OutputVariables[0,112]	AT %QB."KUKA1_KRC5_ProfiNet_6_0".Module001_8_digital_outputs_O_112;
	::OutputVariables[0,113]	AT %QB."KUKA1_KRC5_ProfiNet_6_0".Module001_8_digital_outputs_O_113;
	::OutputVariables[0,114]	AT %QB."KUKA1_KRC5_ProfiNet_6_0".Module001_8_digital_outputs_O_114;
	::OutputVariables[0,115]	AT %QB."KUKA1_KRC5_ProfiNet_6_0".Module001_8_digital_outputs_O_115;
	::OutputVariables[0,116]	AT %QB."KUKA1_KRC5_ProfiNet_6_0".Module001_8_digital_outputs_O_116;
	::OutputVariables[0,117]	AT %QB."KUKA1_KRC5_ProfiNet_6_0".Module001_8_digital_outputs_O_117;
	::OutputVariables[0,118]	AT %QB."KUKA1_KRC5_ProfiNet_6_0".Module001_8_digital_outputs_O_118;
	::OutputVariables[0,119]	AT %QB."KUKA1_KRC5_ProfiNet_6_0".Module001_8_digital_outputs_O_119;
	::OutputVariables[0,120]	AT %QB."KUKA1_KRC5_ProfiNet_6_0".Module001_8_digital_outputs_O_120;
	::OutputVariables[0,121]	AT %QB."KUKA1_KRC5_ProfiNet_6_0".Module001_8_digital_outputs_O_121;
	::OutputVariables[0,122]	AT %QB."KUKA1_KRC5_ProfiNet_6_0".Module001_8_digital_outputs_O_122;
	::OutputVariables[0,123]	AT %QB."KUKA1_KRC5_ProfiNet_6_0".Module001_8_digital_outputs_O_123;
	::OutputVariables[0,124]	AT %QB."KUKA1_KRC5_ProfiNet_6_0".Module001_8_digital_outputs_O_124;
	::OutputVariables[0,125]	AT %QB."KUKA1_KRC5_ProfiNet_6_0".Module001_8_digital_outputs_O_125;
	::OutputVariables[0,126]	AT %QB."KUKA1_KRC5_ProfiNet_6_0".Module001_8_digital_outputs_O_126;
	::OutputVariables[0,127]	AT %QB."KUKA1_KRC5_ProfiNet_6_0".Module001_8_digital_outputs_O_127;
	::OutputVariables[0,128]	AT %QB."KUKA1_KRC5_ProfiNet_6_0".Module001_8_digital_outputs_O_128;
	::OutputVariables[0,129]	AT %QB."KUKA1_KRC5_ProfiNet_6_0".Module001_8_digital_outputs_O_129;
	::OutputVariables[0,130]	AT %QB."KUKA1_KRC5_ProfiNet_6_0".Module001_8_digital_outputs_O_130;
	::OutputVariables[0,131]	AT %QB."KUKA1_KRC5_ProfiNet_6_0".Module001_8_digital_outputs_O_131;
	::OutputVariables[0,132]	AT %QB."KUKA1_KRC5_ProfiNet_6_0".Module001_8_digital_outputs_O_132;
	::OutputVariables[0,133]	AT %QB."KUKA1_KRC5_ProfiNet_6_0".Module001_8_digital_outputs_O_133;
	::OutputVariables[0,134]	AT %QB."KUKA1_KRC5_ProfiNet_6_0".Module001_8_digital_outputs_O_134;
	::OutputVariables[0,135]	AT %QB."KUKA1_KRC5_ProfiNet_6_0".Module001_8_digital_outputs_O_135;
	::OutputVariables[0,136]	AT %QB."KUKA1_KRC5_ProfiNet_6_0".Module001_8_digital_outputs_O_136;
	::OutputVariables[0,137]	AT %QB."KUKA1_KRC5_ProfiNet_6_0".Module001_8_digital_outputs_O_137;
	::OutputVariables[0,138]	AT %QB."KUKA1_KRC5_ProfiNet_6_0".Module001_8_digital_outputs_O_138;
	::OutputVariables[0,139]	AT %QB."KUKA1_KRC5_ProfiNet_6_0".Module001_8_digital_outputs_O_139;
	::OutputVariables[0,140]	AT %QB."KUKA1_KRC5_ProfiNet_6_0".Module001_8_digital_outputs_O_140;
	::OutputVariables[0,141]	AT %QB."KUKA1_KRC5_ProfiNet_6_0".Module001_8_digital_outputs_O_141;
	::OutputVariables[0,142]	AT %QB."KUKA1_KRC5_ProfiNet_6_0".Module001_8_digital_outputs_O_142;
	::OutputVariables[0,143]	AT %QB."KUKA1_KRC5_ProfiNet_6_0".Module001_8_digital_outputs_O_143;
	::OutputVariables[0,144]	AT %QB."KUKA1_KRC5_ProfiNet_6_0".Module001_8_digital_outputs_O_144;
	::OutputVariables[0,145]	AT %QB."KUKA1_KRC5_ProfiNet_6_0".Module001_8_digital_outputs_O_145;
	::OutputVariables[0,146]	AT %QB."KUKA1_KRC5_ProfiNet_6_0".Module001_8_digital_outputs_O_146;
	::OutputVariables[0,147]	AT %QB."KUKA1_KRC5_ProfiNet_6_0".Module001_8_digital_outputs_O_147;
	::OutputVariables[0,148]	AT %QB."KUKA1_KRC5_ProfiNet_6_0".Module001_8_digital_outputs_O_148;
	::OutputVariables[0,149]	AT %QB."KUKA1_KRC5_ProfiNet_6_0".Module001_8_digital_outputs_O_149;
	::OutputVariables[0,150]	AT %QB."KUKA1_KRC5_ProfiNet_6_0".Module001_8_digital_outputs_O_150;
	::OutputVariables[0,151]	AT %QB."KUKA1_KRC5_ProfiNet_6_0".Module001_8_digital_outputs_O_151;
	::OutputVariables[0,152]	AT %QB."KUKA1_KRC5_ProfiNet_6_0".Module001_8_digital_outputs_O_152;
	::OutputVariables[0,153]	AT %QB."KUKA1_KRC5_ProfiNet_6_0".Module001_8_digital_outputs_O_153;
	::OutputVariables[0,154]	AT %QB."KUKA1_KRC5_ProfiNet_6_0".Module001_8_digital_outputs_O_154;
	::OutputVariables[0,155]	AT %QB."KUKA1_KRC5_ProfiNet_6_0".Module001_8_digital_outputs_O_155;
	::OutputVariables[0,156]	AT %QB."KUKA1_KRC5_ProfiNet_6_0".Module001_8_digital_outputs_O_156;
	::OutputVariables[0,157]	AT %QB."KUKA1_KRC5_ProfiNet_6_0".Module001_8_digital_outputs_O_157;
	::OutputVariables[0,158]	AT %QB."KUKA1_KRC5_ProfiNet_6_0".Module001_8_digital_outputs_O_158;
	::OutputVariables[0,159]	AT %QB."KUKA1_KRC5_ProfiNet_6_0".Module001_8_digital_outputs_O_159;
	::OutputVariables[0,160]	AT %QB."KUKA1_KRC5_ProfiNet_6_0".Module001_8_digital_outputs_O_160;
	::OutputVariables[0,161]	AT %QB."KUKA1_KRC5_ProfiNet_6_0".Module001_8_digital_outputs_O_161;
	::OutputVariables[0,162]	AT %QB."KUKA1_KRC5_ProfiNet_6_0".Module001_8_digital_outputs_O_162;
	::OutputVariables[0,163]	AT %QB."KUKA1_KRC5_ProfiNet_6_0".Module001_8_digital_outputs_O_163;
	::OutputVariables[0,164]	AT %QB."KUKA1_KRC5_ProfiNet_6_0".Module001_8_digital_outputs_O_164;
	::OutputVariables[0,165]	AT %QB."KUKA1_KRC5_ProfiNet_6_0".Module001_8_digital_outputs_O_165;
	::OutputVariables[0,166]	AT %QB."KUKA1_KRC5_ProfiNet_6_0".Module001_8_digital_outputs_O_166;
	::OutputVariables[0,167]	AT %QB."KUKA1_KRC5_ProfiNet_6_0".Module001_8_digital_outputs_O_167;
	::OutputVariables[0,168]	AT %QB."KUKA1_KRC5_ProfiNet_6_0".Module001_8_digital_outputs_O_168;
	::OutputVariables[0,169]	AT %QB."KUKA1_KRC5_ProfiNet_6_0".Module001_8_digital_outputs_O_169;
	::OutputVariables[0,170]	AT %QB."KUKA1_KRC5_ProfiNet_6_0".Module001_8_digital_outputs_O_170;
	::OutputVariables[0,171]	AT %QB."KUKA1_KRC5_ProfiNet_6_0".Module001_8_digital_outputs_O_171;
	::OutputVariables[0,172]	AT %QB."KUKA1_KRC5_ProfiNet_6_0".Module001_8_digital_outputs_O_172;
	::OutputVariables[0,173]	AT %QB."KUKA1_KRC5_ProfiNet_6_0".Module001_8_digital_outputs_O_173;
	::OutputVariables[0,174]	AT %QB."KUKA1_KRC5_ProfiNet_6_0".Module001_8_digital_outputs_O_174;
	::OutputVariables[0,175]	AT %QB."KUKA1_KRC5_ProfiNet_6_0".Module001_8_digital_outputs_O_175;
	::OutputVariables[0,176]	AT %QB."KUKA1_KRC5_ProfiNet_6_0".Module001_8_digital_outputs_O_176;
	::OutputVariables[0,177]	AT %QB."KUKA1_KRC5_ProfiNet_6_0".Module001_8_digital_outputs_O_177;
	::OutputVariables[0,178]	AT %QB."KUKA1_KRC5_ProfiNet_6_0".Module001_8_digital_outputs_O_178;
	::OutputVariables[0,179]	AT %QB."KUKA1_KRC5_ProfiNet_6_0".Module001_8_digital_outputs_O_179;
	::OutputVariables[0,180]	AT %QB."KUKA1_KRC5_ProfiNet_6_0".Module001_8_digital_outputs_O_180;
	::OutputVariables[0,181]	AT %QB."KUKA1_KRC5_ProfiNet_6_0".Module001_8_digital_outputs_O_181;
	::OutputVariables[0,182]	AT %QB."KUKA1_KRC5_ProfiNet_6_0".Module001_8_digital_outputs_O_182;
	::OutputVariables[0,183]	AT %QB."KUKA1_KRC5_ProfiNet_6_0".Module001_8_digital_outputs_O_183;
	::OutputVariables[0,184]	AT %QB."KUKA1_KRC5_ProfiNet_6_0".Module001_8_digital_outputs_O_184;
	::OutputVariables[0,185]	AT %QB."KUKA1_KRC5_ProfiNet_6_0".Module001_8_digital_outputs_O_185;
	::OutputVariables[0,186]	AT %QB."KUKA1_KRC5_ProfiNet_6_0".Module001_8_digital_outputs_O_186;
	::OutputVariables[0,187]	AT %QB."KUKA1_KRC5_ProfiNet_6_0".Module001_8_digital_outputs_O_187;
	::OutputVariables[0,188]	AT %QB."KUKA1_KRC5_ProfiNet_6_0".Module001_8_digital_outputs_O_188;
	::OutputVariables[0,189]	AT %QB."KUKA1_KRC5_ProfiNet_6_0".Module001_8_digital_outputs_O_189;
	::OutputVariables[0,190]	AT %QB."KUKA1_KRC5_ProfiNet_6_0".Module001_8_digital_outputs_O_190;
	::OutputVariables[0,191]	AT %QB."KUKA1_KRC5_ProfiNet_6_0".Module001_8_digital_outputs_O_191;
	::OutputVariables[0,192]	AT %QB."KUKA1_KRC5_ProfiNet_6_0".Module001_8_digital_outputs_O_192;
	::OutputVariables[0,193]	AT %QB."KUKA1_KRC5_ProfiNet_6_0".Module001_8_digital_outputs_O_193;
	::OutputVariables[0,194]	AT %QB."KUKA1_KRC5_ProfiNet_6_0".Module001_8_digital_outputs_O_194;
	::OutputVariables[0,195]	AT %QB."KUKA1_KRC5_ProfiNet_6_0".Module001_8_digital_outputs_O_195;
	::OutputVariables[0,196]	AT %QB."KUKA1_KRC5_ProfiNet_6_0".Module001_8_digital_outputs_O_196;
	::OutputVariables[0,197]	AT %QB."KUKA1_KRC5_ProfiNet_6_0".Module001_8_digital_outputs_O_197;
	::OutputVariables[0,198]	AT %QB."KUKA1_KRC5_ProfiNet_6_0".Module001_8_digital_outputs_O_198;
	::OutputVariables[0,199]	AT %QB."KUKA1_KRC5_ProfiNet_6_0".Module001_8_digital_outputs_O_199;
	::OutputVariables[0,200]	AT %QB."KUKA1_KRC5_ProfiNet_6_0".Module001_8_digital_outputs_O_200;
	::OutputVariables[0,201]	AT %QB."KUKA1_KRC5_ProfiNet_6_0".Module001_8_digital_outputs_O_201;
	::OutputVariables[0,202]	AT %QB."KUKA1_KRC5_ProfiNet_6_0".Module001_8_digital_outputs_O_202;
	::OutputVariables[0,203]	AT %QB."KUKA1_KRC5_ProfiNet_6_0".Module001_8_digital_outputs_O_203;
	::OutputVariables[0,204]	AT %QB."KUKA1_KRC5_ProfiNet_6_0".Module001_8_digital_outputs_O_204;
	::OutputVariables[0,205]	AT %QB."KUKA1_KRC5_ProfiNet_6_0".Module001_8_digital_outputs_O_205;
	::OutputVariables[0,206]	AT %QB."KUKA1_KRC5_ProfiNet_6_0".Module001_8_digital_outputs_O_206;
	::OutputVariables[0,207]	AT %QB."KUKA1_KRC5_ProfiNet_6_0".Module001_8_digital_outputs_O_207;
	::OutputVariables[0,208]	AT %QB."KUKA1_KRC5_ProfiNet_6_0".Module001_8_digital_outputs_O_208;
	::OutputVariables[0,209]	AT %QB."KUKA1_KRC5_ProfiNet_6_0".Module001_8_digital_outputs_O_209;
	::OutputVariables[0,210]	AT %QB."KUKA1_KRC5_ProfiNet_6_0".Module001_8_digital_outputs_O_210;
	::OutputVariables[0,211]	AT %QB."KUKA1_KRC5_ProfiNet_6_0".Module001_8_digital_outputs_O_211;
	::OutputVariables[0,212]	AT %QB."KUKA1_KRC5_ProfiNet_6_0".Module001_8_digital_outputs_O_212;
	::OutputVariables[0,213]	AT %QB."KUKA1_KRC5_ProfiNet_6_0".Module001_8_digital_outputs_O_213;
	::OutputVariables[0,214]	AT %QB."KUKA1_KRC5_ProfiNet_6_0".Module001_8_digital_outputs_O_214;
	::OutputVariables[0,215]	AT %QB."KUKA1_KRC5_ProfiNet_6_0".Module001_8_digital_outputs_O_215;
	::OutputVariables[0,216]	AT %QB."KUKA1_KRC5_ProfiNet_6_0".Module001_8_digital_outputs_O_216;
	::OutputVariables[0,217]	AT %QB."KUKA1_KRC5_ProfiNet_6_0".Module001_8_digital_outputs_O_217;
	::OutputVariables[0,218]	AT %QB."KUKA1_KRC5_ProfiNet_6_0".Module001_8_digital_outputs_O_218;
	::OutputVariables[0,219]	AT %QB."KUKA1_KRC5_ProfiNet_6_0".Module001_8_digital_outputs_O_219;
	::OutputVariables[0,220]	AT %QB."KUKA1_KRC5_ProfiNet_6_0".Module001_8_digital_outputs_O_220;
	::OutputVariables[0,221]	AT %QB."KUKA1_KRC5_ProfiNet_6_0".Module001_8_digital_outputs_O_221;
	::OutputVariables[0,222]	AT %QB."KUKA1_KRC5_ProfiNet_6_0".Module001_8_digital_outputs_O_222;
	::OutputVariables[0,223]	AT %QB."KUKA1_KRC5_ProfiNet_6_0".Module001_8_digital_outputs_O_223;
	::OutputVariables[0,224]	AT %QB."KUKA1_KRC5_ProfiNet_6_0".Module001_8_digital_outputs_O_224;
	::OutputVariables[0,225]	AT %QB."KUKA1_KRC5_ProfiNet_6_0".Module001_8_digital_outputs_O_225;
	::OutputVariables[0,226]	AT %QB."KUKA1_KRC5_ProfiNet_6_0".Module001_8_digital_outputs_O_226;
	::OutputVariables[0,227]	AT %QB."KUKA1_KRC5_ProfiNet_6_0".Module001_8_digital_outputs_O_227;
	::OutputVariables[0,228]	AT %QB."KUKA1_KRC5_ProfiNet_6_0".Module001_8_digital_outputs_O_228;
	::OutputVariables[0,229]	AT %QB."KUKA1_KRC5_ProfiNet_6_0".Module001_8_digital_outputs_O_229;
	::OutputVariables[0,230]	AT %QB."KUKA1_KRC5_ProfiNet_6_0".Module001_8_digital_outputs_O_230;
	::OutputVariables[0,231]	AT %QB."KUKA1_KRC5_ProfiNet_6_0".Module001_8_digital_outputs_O_231;
	::OutputVariables[0,232]	AT %QB."KUKA1_KRC5_ProfiNet_6_0".Module001_8_digital_outputs_O_232;
	::OutputVariables[0,233]	AT %QB."KUKA1_KRC5_ProfiNet_6_0".Module001_8_digital_outputs_O_233;
	::OutputVariables[0,234]	AT %QB."KUKA1_KRC5_ProfiNet_6_0".Module001_8_digital_outputs_O_234;
	::OutputVariables[0,235]	AT %QB."KUKA1_KRC5_ProfiNet_6_0".Module001_8_digital_outputs_O_235;
	::OutputVariables[0,236]	AT %QB."KUKA1_KRC5_ProfiNet_6_0".Module001_8_digital_outputs_O_236;
	::OutputVariables[0,237]	AT %QB."KUKA1_KRC5_ProfiNet_6_0".Module001_8_digital_outputs_O_237;
	::OutputVariables[0,238]	AT %QB."KUKA1_KRC5_ProfiNet_6_0".Module001_8_digital_outputs_O_238;
	::OutputVariables[0,239]	AT %QB."KUKA1_KRC5_ProfiNet_6_0".Module001_8_digital_outputs_O_239;
	::OutputVariables[0,240]	AT %QB."KUKA1_KRC5_ProfiNet_6_0".Module001_8_digital_outputs_O_240;
	::OutputVariables[0,241]	AT %QB."KUKA1_KRC5_ProfiNet_6_0".Module001_8_digital_outputs_O_241;
	::OutputVariables[0,242]	AT %QB."KUKA1_KRC5_ProfiNet_6_0".Module001_8_digital_outputs_O_242;
	::OutputVariables[0,243]	AT %QB."KUKA1_KRC5_ProfiNet_6_0".Module001_8_digital_outputs_O_243;
	::OutputVariables[0,244]	AT %QB."KUKA1_KRC5_ProfiNet_6_0".Module001_8_digital_outputs_O_244;
	::OutputVariables[0,245]	AT %QB."KUKA1_KRC5_ProfiNet_6_0".Module001_8_digital_outputs_O_245;
	::OutputVariables[0,246]	AT %QB."KUKA1_KRC5_ProfiNet_6_0".Module001_8_digital_outputs_O_246;
	::OutputVariables[0,247]	AT %QB."KUKA1_KRC5_ProfiNet_6_0".Module001_8_digital_outputs_O_247;
	::OutputVariables[0,248]	AT %QB."KUKA1_KRC5_ProfiNet_6_0".Module001_8_digital_outputs_O_248;
	::OutputVariables[0,249]	AT %QB."KUKA1_KRC5_ProfiNet_6_0".Module001_8_digital_outputs_O_249;
	::OutputVariables[0,250]	AT %QB."KUKA1_KRC5_ProfiNet_6_0".Module001_8_digital_outputs_O_250;
	::OutputVariables[0,251]	AT %QB."KUKA1_KRC5_ProfiNet_6_0".Module001_8_digital_outputs_O_251;
	::OutputVariables[0,252]	AT %QB."KUKA1_KRC5_ProfiNet_6_0".Module001_8_digital_outputs_O_252;
	::OutputVariables[0,253]	AT %QB."KUKA1_KRC5_ProfiNet_6_0".Module001_8_digital_outputs_O_253;

	(*________________________________________*)
	(*_____________KUKA2 Mappings_____________*)
	(*________________________________________*)
	::InputVariables[1,0] AT %IB."KUKA2_KRC4_ProfiNet_5_0".Module001_8_digital_inputs_I_00;
	::InputVariables[1,1] AT %IB."KUKA2_KRC4_ProfiNet_5_0".Module001_8_digital_inputs_I_01;
	::InputVariables[1,2] AT %IB."KUKA2_KRC4_ProfiNet_5_0".Module001_8_digital_inputs_I_02;
	::InputVariables[1,3] AT %IB."KUKA2_KRC4_ProfiNet_5_0".Module001_8_digital_inputs_I_03;
	::InputVariables[1,4] AT %IB."KUKA2_KRC4_ProfiNet_5_0".Module001_8_digital_inputs_I_04;
	::InputVariables[1,5] AT %IB."KUKA2_KRC4_ProfiNet_5_0".Module001_8_digital_inputs_I_05;
	::InputVariables[1,6] AT %IB."KUKA2_KRC4_ProfiNet_5_0".Module001_8_digital_inputs_I_06;
	::InputVariables[1,7] AT %IB."KUKA2_KRC4_ProfiNet_5_0".Module001_8_digital_inputs_I_07;
	::InputVariables[1,8] AT %IB."KUKA2_KRC4_ProfiNet_5_0".Module001_8_digital_inputs_I_08;
	::InputVariables[1,9] AT %IB."KUKA2_KRC4_ProfiNet_5_0".Module001_8_digital_inputs_I_09;
	::InputVariables[1,10] AT %IB."KUKA2_KRC4_ProfiNet_5_0".Module001_8_digital_inputs_I_10;
	::InputVariables[1,11] AT %IB."KUKA2_KRC4_ProfiNet_5_0".Module001_8_digital_inputs_I_11;
	::InputVariables[1,12] AT %IB."KUKA2_KRC4_ProfiNet_5_0".Module001_8_digital_inputs_I_12;
	::InputVariables[1,13] AT %IB."KUKA2_KRC4_ProfiNet_5_0".Module001_8_digital_inputs_I_13;
	::InputVariables[1,14] AT %IB."KUKA2_KRC4_ProfiNet_5_0".Module001_8_digital_inputs_I_14;
	::InputVariables[1,15] AT %IB."KUKA2_KRC4_ProfiNet_5_0".Module001_8_digital_inputs_I_15;
	::InputVariables[1,16] AT %IB."KUKA2_KRC4_ProfiNet_5_0".Module001_8_digital_inputs_I_16;
	::InputVariables[1,17] AT %IB."KUKA2_KRC4_ProfiNet_5_0".Module001_8_digital_inputs_I_17;
	::InputVariables[1,18] AT %IB."KUKA2_KRC4_ProfiNet_5_0".Module001_8_digital_inputs_I_18;
	::InputVariables[1,19] AT %IB."KUKA2_KRC4_ProfiNet_5_0".Module001_8_digital_inputs_I_19;
	::InputVariables[1,20] AT %IB."KUKA2_KRC4_ProfiNet_5_0".Module001_8_digital_inputs_I_20;
	::InputVariables[1,21] AT %IB."KUKA2_KRC4_ProfiNet_5_0".Module001_8_digital_inputs_I_21;
	::InputVariables[1,22] AT %IB."KUKA2_KRC4_ProfiNet_5_0".Module001_8_digital_inputs_I_22;
	::InputVariables[1,23] AT %IB."KUKA2_KRC4_ProfiNet_5_0".Module001_8_digital_inputs_I_23;
	::InputVariables[1,24] AT %IB."KUKA2_KRC4_ProfiNet_5_0".Module001_8_digital_inputs_I_24;
	::InputVariables[1,25] AT %IB."KUKA2_KRC4_ProfiNet_5_0".Module001_8_digital_inputs_I_25;
	::InputVariables[1,26] AT %IB."KUKA2_KRC4_ProfiNet_5_0".Module001_8_digital_inputs_I_26;
	::InputVariables[1,27] AT %IB."KUKA2_KRC4_ProfiNet_5_0".Module001_8_digital_inputs_I_27;
	::InputVariables[1,28] AT %IB."KUKA2_KRC4_ProfiNet_5_0".Module001_8_digital_inputs_I_28;
	::InputVariables[1,29] AT %IB."KUKA2_KRC4_ProfiNet_5_0".Module001_8_digital_inputs_I_29;
	::InputVariables[1,30] AT %IB."KUKA2_KRC4_ProfiNet_5_0".Module001_8_digital_inputs_I_30;
	::InputVariables[1,31] AT %IB."KUKA2_KRC4_ProfiNet_5_0".Module001_8_digital_inputs_I_31;
	::InputVariables[1,32] AT %IB."KUKA2_KRC4_ProfiNet_5_0".Module001_8_digital_inputs_I_32;
	::InputVariables[1,33] AT %IB."KUKA2_KRC4_ProfiNet_5_0".Module001_8_digital_inputs_I_33;
	::InputVariables[1,34] AT %IB."KUKA2_KRC4_ProfiNet_5_0".Module001_8_digital_inputs_I_34;
	::InputVariables[1,35] AT %IB."KUKA2_KRC4_ProfiNet_5_0".Module001_8_digital_inputs_I_35;
	::InputVariables[1,36] AT %IB."KUKA2_KRC4_ProfiNet_5_0".Module001_8_digital_inputs_I_36;
	::InputVariables[1,37] AT %IB."KUKA2_KRC4_ProfiNet_5_0".Module001_8_digital_inputs_I_37;
	::InputVariables[1,38] AT %IB."KUKA2_KRC4_ProfiNet_5_0".Module001_8_digital_inputs_I_38;
	::InputVariables[1,39] AT %IB."KUKA2_KRC4_ProfiNet_5_0".Module001_8_digital_inputs_I_39;
	::InputVariables[1,40] AT %IB."KUKA2_KRC4_ProfiNet_5_0".Module001_8_digital_inputs_I_40;
	::InputVariables[1,41] AT %IB."KUKA2_KRC4_ProfiNet_5_0".Module001_8_digital_inputs_I_41;
	::InputVariables[1,42] AT %IB."KUKA2_KRC4_ProfiNet_5_0".Module001_8_digital_inputs_I_42;
	::InputVariables[1,43] AT %IB."KUKA2_KRC4_ProfiNet_5_0".Module001_8_digital_inputs_I_43;
	::InputVariables[1,44] AT %IB."KUKA2_KRC4_ProfiNet_5_0".Module001_8_digital_inputs_I_44;
	::InputVariables[1,45] AT %IB."KUKA2_KRC4_ProfiNet_5_0".Module001_8_digital_inputs_I_45;
	::InputVariables[1,46] AT %IB."KUKA2_KRC4_ProfiNet_5_0".Module001_8_digital_inputs_I_46;
	::InputVariables[1,47] AT %IB."KUKA2_KRC4_ProfiNet_5_0".Module001_8_digital_inputs_I_47;
	::InputVariables[1,48] AT %IB."KUKA2_KRC4_ProfiNet_5_0".Module001_8_digital_inputs_I_48;
	::InputVariables[1,49] AT %IB."KUKA2_KRC4_ProfiNet_5_0".Module001_8_digital_inputs_I_49;
	::InputVariables[1,50] AT %IB."KUKA2_KRC4_ProfiNet_5_0".Module001_8_digital_inputs_I_50;
	::InputVariables[1,51] AT %IB."KUKA2_KRC4_ProfiNet_5_0".Module001_8_digital_inputs_I_51;
	::InputVariables[1,52] AT %IB."KUKA2_KRC4_ProfiNet_5_0".Module001_8_digital_inputs_I_52;
	::InputVariables[1,53] AT %IB."KUKA2_KRC4_ProfiNet_5_0".Module001_8_digital_inputs_I_53;
	::InputVariables[1,54] AT %IB."KUKA2_KRC4_ProfiNet_5_0".Module001_8_digital_inputs_I_54;
	::InputVariables[1,55] AT %IB."KUKA2_KRC4_ProfiNet_5_0".Module001_8_digital_inputs_I_55;
	::InputVariables[1,56] AT %IB."KUKA2_KRC4_ProfiNet_5_0".Module001_8_digital_inputs_I_56;
	::InputVariables[1,57] AT %IB."KUKA2_KRC4_ProfiNet_5_0".Module001_8_digital_inputs_I_57;
	::InputVariables[1,58] AT %IB."KUKA2_KRC4_ProfiNet_5_0".Module001_8_digital_inputs_I_58;
	::InputVariables[1,59] AT %IB."KUKA2_KRC4_ProfiNet_5_0".Module001_8_digital_inputs_I_59;
	::InputVariables[1,60] AT %IB."KUKA2_KRC4_ProfiNet_5_0".Module001_8_digital_inputs_I_60;
	::InputVariables[1,61] AT %IB."KUKA2_KRC4_ProfiNet_5_0".Module001_8_digital_inputs_I_61;
	::InputVariables[1,62] AT %IB."KUKA2_KRC4_ProfiNet_5_0".Module001_8_digital_inputs_I_62;
	::InputVariables[1,63] AT %IB."KUKA2_KRC4_ProfiNet_5_0".Module001_8_digital_inputs_I_63;
	::InputVariables[1,64] AT %IB."KUKA2_KRC4_ProfiNet_5_0".Module001_8_digital_inputs_I_64;
	::InputVariables[1,65] AT %IB."KUKA2_KRC4_ProfiNet_5_0".Module001_8_digital_inputs_I_65;
	::InputVariables[1,66] AT %IB."KUKA2_KRC4_ProfiNet_5_0".Module001_8_digital_inputs_I_66;
	::InputVariables[1,67] AT %IB."KUKA2_KRC4_ProfiNet_5_0".Module001_8_digital_inputs_I_67;
	::InputVariables[1,68] AT %IB."KUKA2_KRC4_ProfiNet_5_0".Module001_8_digital_inputs_I_68;
	::InputVariables[1,69] AT %IB."KUKA2_KRC4_ProfiNet_5_0".Module001_8_digital_inputs_I_69;
	::InputVariables[1,70] AT %IB."KUKA2_KRC4_ProfiNet_5_0".Module001_8_digital_inputs_I_70;
	::InputVariables[1,71] AT %IB."KUKA2_KRC4_ProfiNet_5_0".Module001_8_digital_inputs_I_71;
	::InputVariables[1,72] AT %IB."KUKA2_KRC4_ProfiNet_5_0".Module001_8_digital_inputs_I_72;
	::InputVariables[1,73] AT %IB."KUKA2_KRC4_ProfiNet_5_0".Module001_8_digital_inputs_I_73;
	::InputVariables[1,74] AT %IB."KUKA2_KRC4_ProfiNet_5_0".Module001_8_digital_inputs_I_74;
	::InputVariables[1,75] AT %IB."KUKA2_KRC4_ProfiNet_5_0".Module001_8_digital_inputs_I_75;
	::InputVariables[1,76] AT %IB."KUKA2_KRC4_ProfiNet_5_0".Module001_8_digital_inputs_I_76;
	::InputVariables[1,77] AT %IB."KUKA2_KRC4_ProfiNet_5_0".Module001_8_digital_inputs_I_77;
	::InputVariables[1,78] AT %IB."KUKA2_KRC4_ProfiNet_5_0".Module001_8_digital_inputs_I_78;
	::InputVariables[1,79] AT %IB."KUKA2_KRC4_ProfiNet_5_0".Module001_8_digital_inputs_I_79;
	::InputVariables[1,80] AT %IB."KUKA2_KRC4_ProfiNet_5_0".Module001_8_digital_inputs_I_80;
	::InputVariables[1,81] AT %IB."KUKA2_KRC4_ProfiNet_5_0".Module001_8_digital_inputs_I_81;
	::InputVariables[1,82] AT %IB."KUKA2_KRC4_ProfiNet_5_0".Module001_8_digital_inputs_I_82;
	::InputVariables[1,83] AT %IB."KUKA2_KRC4_ProfiNet_5_0".Module001_8_digital_inputs_I_83;
	::InputVariables[1,84] AT %IB."KUKA2_KRC4_ProfiNet_5_0".Module001_8_digital_inputs_I_84;
	::InputVariables[1,85] AT %IB."KUKA2_KRC4_ProfiNet_5_0".Module001_8_digital_inputs_I_85;
	::InputVariables[1,86] AT %IB."KUKA2_KRC4_ProfiNet_5_0".Module001_8_digital_inputs_I_86;
	::InputVariables[1,87] AT %IB."KUKA2_KRC4_ProfiNet_5_0".Module001_8_digital_inputs_I_87;
	::InputVariables[1,88] AT %IB."KUKA2_KRC4_ProfiNet_5_0".Module001_8_digital_inputs_I_88;
	::InputVariables[1,89] AT %IB."KUKA2_KRC4_ProfiNet_5_0".Module001_8_digital_inputs_I_89;
	::InputVariables[1,90] AT %IB."KUKA2_KRC4_ProfiNet_5_0".Module001_8_digital_inputs_I_90;
	::InputVariables[1,91] AT %IB."KUKA2_KRC4_ProfiNet_5_0".Module001_8_digital_inputs_I_91;
	::InputVariables[1,92] AT %IB."KUKA2_KRC4_ProfiNet_5_0".Module001_8_digital_inputs_I_92;
	::InputVariables[1,93] AT %IB."KUKA2_KRC4_ProfiNet_5_0".Module001_8_digital_inputs_I_93;
	::InputVariables[1,94] AT %IB."KUKA2_KRC4_ProfiNet_5_0".Module001_8_digital_inputs_I_94;
	::InputVariables[1,95] AT %IB."KUKA2_KRC4_ProfiNet_5_0".Module001_8_digital_inputs_I_95;
	::InputVariables[1,96] AT %IB."KUKA2_KRC4_ProfiNet_5_0".Module001_8_digital_inputs_I_96;
	::InputVariables[1,97] AT %IB."KUKA2_KRC4_ProfiNet_5_0".Module001_8_digital_inputs_I_97;
	::InputVariables[1,98] AT %IB."KUKA2_KRC4_ProfiNet_5_0".Module001_8_digital_inputs_I_98;
	::InputVariables[1,99] AT %IB."KUKA2_KRC4_ProfiNet_5_0".Module001_8_digital_inputs_I_99;
	::InputVariables[1,100] AT %IB."KUKA2_KRC4_ProfiNet_5_0".Module001_8_digital_inputs_I_100;
	::InputVariables[1,101] AT %IB."KUKA2_KRC4_ProfiNet_5_0".Module001_8_digital_inputs_I_101;
	::InputVariables[1,102] AT %IB."KUKA2_KRC4_ProfiNet_5_0".Module001_8_digital_inputs_I_102;
	::InputVariables[1,103] AT %IB."KUKA2_KRC4_ProfiNet_5_0".Module001_8_digital_inputs_I_103;
	::InputVariables[1,104] AT %IB."KUKA2_KRC4_ProfiNet_5_0".Module001_8_digital_inputs_I_104;
	::InputVariables[1,105] AT %IB."KUKA2_KRC4_ProfiNet_5_0".Module001_8_digital_inputs_I_105;
	::InputVariables[1,106] AT %IB."KUKA2_KRC4_ProfiNet_5_0".Module001_8_digital_inputs_I_106;
	::InputVariables[1,107] AT %IB."KUKA2_KRC4_ProfiNet_5_0".Module001_8_digital_inputs_I_107;
	::InputVariables[1,108] AT %IB."KUKA2_KRC4_ProfiNet_5_0".Module001_8_digital_inputs_I_108;
	::InputVariables[1,109] AT %IB."KUKA2_KRC4_ProfiNet_5_0".Module001_8_digital_inputs_I_109;
	::InputVariables[1,110] AT %IB."KUKA2_KRC4_ProfiNet_5_0".Module001_8_digital_inputs_I_110;
	::InputVariables[1,111] AT %IB."KUKA2_KRC4_ProfiNet_5_0".Module001_8_digital_inputs_I_111;
	::InputVariables[1,112] AT %IB."KUKA2_KRC4_ProfiNet_5_0".Module001_8_digital_inputs_I_112;
	::InputVariables[1,113] AT %IB."KUKA2_KRC4_ProfiNet_5_0".Module001_8_digital_inputs_I_113;
	::InputVariables[1,114] AT %IB."KUKA2_KRC4_ProfiNet_5_0".Module001_8_digital_inputs_I_114;
	::InputVariables[1,115] AT %IB."KUKA2_KRC4_ProfiNet_5_0".Module001_8_digital_inputs_I_115;
	::InputVariables[1,116] AT %IB."KUKA2_KRC4_ProfiNet_5_0".Module001_8_digital_inputs_I_116;
	::InputVariables[1,117] AT %IB."KUKA2_KRC4_ProfiNet_5_0".Module001_8_digital_inputs_I_117;
	::InputVariables[1,118] AT %IB."KUKA2_KRC4_ProfiNet_5_0".Module001_8_digital_inputs_I_118;
	::InputVariables[1,119] AT %IB."KUKA2_KRC4_ProfiNet_5_0".Module001_8_digital_inputs_I_119;
	::InputVariables[1,120] AT %IB."KUKA2_KRC4_ProfiNet_5_0".Module001_8_digital_inputs_I_120;
	::InputVariables[1,121] AT %IB."KUKA2_KRC4_ProfiNet_5_0".Module001_8_digital_inputs_I_121;
	::InputVariables[1,122] AT %IB."KUKA2_KRC4_ProfiNet_5_0".Module001_8_digital_inputs_I_122;
	::InputVariables[1,123] AT %IB."KUKA2_KRC4_ProfiNet_5_0".Module001_8_digital_inputs_I_123;
	::InputVariables[1,124] AT %IB."KUKA2_KRC4_ProfiNet_5_0".Module001_8_digital_inputs_I_124;
	::InputVariables[1,125] AT %IB."KUKA2_KRC4_ProfiNet_5_0".Module001_8_digital_inputs_I_125;
	::InputVariables[1,126] AT %IB."KUKA2_KRC4_ProfiNet_5_0".Module001_8_digital_inputs_I_126;
	::InputVariables[1,127] AT %IB."KUKA2_KRC4_ProfiNet_5_0".Module001_8_digital_inputs_I_127;
	::InputVariables[1,128] AT %IB."KUKA2_KRC4_ProfiNet_5_0".Module001_8_digital_inputs_I_128;
	::InputVariables[1,129] AT %IB."KUKA2_KRC4_ProfiNet_5_0".Module001_8_digital_inputs_I_129;
	::InputVariables[1,130] AT %IB."KUKA2_KRC4_ProfiNet_5_0".Module001_8_digital_inputs_I_130;
	::InputVariables[1,131] AT %IB."KUKA2_KRC4_ProfiNet_5_0".Module001_8_digital_inputs_I_131;
	::InputVariables[1,132] AT %IB."KUKA2_KRC4_ProfiNet_5_0".Module001_8_digital_inputs_I_132;
	::InputVariables[1,133] AT %IB."KUKA2_KRC4_ProfiNet_5_0".Module001_8_digital_inputs_I_133;
	::InputVariables[1,134] AT %IB."KUKA2_KRC4_ProfiNet_5_0".Module001_8_digital_inputs_I_134;
	::InputVariables[1,135] AT %IB."KUKA2_KRC4_ProfiNet_5_0".Module001_8_digital_inputs_I_135;
	::InputVariables[1,136] AT %IB."KUKA2_KRC4_ProfiNet_5_0".Module001_8_digital_inputs_I_136;
	::InputVariables[1,137] AT %IB."KUKA2_KRC4_ProfiNet_5_0".Module001_8_digital_inputs_I_137;
	::InputVariables[1,138] AT %IB."KUKA2_KRC4_ProfiNet_5_0".Module001_8_digital_inputs_I_138;
	::InputVariables[1,139] AT %IB."KUKA2_KRC4_ProfiNet_5_0".Module001_8_digital_inputs_I_139;
	::InputVariables[1,140] AT %IB."KUKA2_KRC4_ProfiNet_5_0".Module001_8_digital_inputs_I_140;
	::InputVariables[1,141] AT %IB."KUKA2_KRC4_ProfiNet_5_0".Module001_8_digital_inputs_I_141;
	::InputVariables[1,142] AT %IB."KUKA2_KRC4_ProfiNet_5_0".Module001_8_digital_inputs_I_142;
	::InputVariables[1,143] AT %IB."KUKA2_KRC4_ProfiNet_5_0".Module001_8_digital_inputs_I_143;
	::InputVariables[1,144] AT %IB."KUKA2_KRC4_ProfiNet_5_0".Module001_8_digital_inputs_I_144;
	::InputVariables[1,145] AT %IB."KUKA2_KRC4_ProfiNet_5_0".Module001_8_digital_inputs_I_145;
	::InputVariables[1,146] AT %IB."KUKA2_KRC4_ProfiNet_5_0".Module001_8_digital_inputs_I_146;
	::InputVariables[1,147] AT %IB."KUKA2_KRC4_ProfiNet_5_0".Module001_8_digital_inputs_I_147;
	::InputVariables[1,148] AT %IB."KUKA2_KRC4_ProfiNet_5_0".Module001_8_digital_inputs_I_148;
	::InputVariables[1,149] AT %IB."KUKA2_KRC4_ProfiNet_5_0".Module001_8_digital_inputs_I_149;
	::InputVariables[1,150] AT %IB."KUKA2_KRC4_ProfiNet_5_0".Module001_8_digital_inputs_I_150;
	::InputVariables[1,151] AT %IB."KUKA2_KRC4_ProfiNet_5_0".Module001_8_digital_inputs_I_151;
	::InputVariables[1,152] AT %IB."KUKA2_KRC4_ProfiNet_5_0".Module001_8_digital_inputs_I_152;
	::InputVariables[1,153] AT %IB."KUKA2_KRC4_ProfiNet_5_0".Module001_8_digital_inputs_I_153;
	::InputVariables[1,154] AT %IB."KUKA2_KRC4_ProfiNet_5_0".Module001_8_digital_inputs_I_154;
	::InputVariables[1,155] AT %IB."KUKA2_KRC4_ProfiNet_5_0".Module001_8_digital_inputs_I_155;
	::InputVariables[1,156] AT %IB."KUKA2_KRC4_ProfiNet_5_0".Module001_8_digital_inputs_I_156;
	::InputVariables[1,157] AT %IB."KUKA2_KRC4_ProfiNet_5_0".Module001_8_digital_inputs_I_157;
	::InputVariables[1,158] AT %IB."KUKA2_KRC4_ProfiNet_5_0".Module001_8_digital_inputs_I_158;
	::InputVariables[1,159] AT %IB."KUKA2_KRC4_ProfiNet_5_0".Module001_8_digital_inputs_I_159;
	::InputVariables[1,160] AT %IB."KUKA2_KRC4_ProfiNet_5_0".Module001_8_digital_inputs_I_160;
	::InputVariables[1,161] AT %IB."KUKA2_KRC4_ProfiNet_5_0".Module001_8_digital_inputs_I_161;
	::InputVariables[1,162] AT %IB."KUKA2_KRC4_ProfiNet_5_0".Module001_8_digital_inputs_I_162;
	::InputVariables[1,163] AT %IB."KUKA2_KRC4_ProfiNet_5_0".Module001_8_digital_inputs_I_163;
	::InputVariables[1,164] AT %IB."KUKA2_KRC4_ProfiNet_5_0".Module001_8_digital_inputs_I_164;
	::InputVariables[1,165] AT %IB."KUKA2_KRC4_ProfiNet_5_0".Module001_8_digital_inputs_I_165;
	::InputVariables[1,166] AT %IB."KUKA2_KRC4_ProfiNet_5_0".Module001_8_digital_inputs_I_166;
	::InputVariables[1,167] AT %IB."KUKA2_KRC4_ProfiNet_5_0".Module001_8_digital_inputs_I_167;
	::InputVariables[1,168] AT %IB."KUKA2_KRC4_ProfiNet_5_0".Module001_8_digital_inputs_I_168;
	::InputVariables[1,169] AT %IB."KUKA2_KRC4_ProfiNet_5_0".Module001_8_digital_inputs_I_169;
	::InputVariables[1,170] AT %IB."KUKA2_KRC4_ProfiNet_5_0".Module001_8_digital_inputs_I_170;
	::InputVariables[1,171] AT %IB."KUKA2_KRC4_ProfiNet_5_0".Module001_8_digital_inputs_I_171;
	::InputVariables[1,172] AT %IB."KUKA2_KRC4_ProfiNet_5_0".Module001_8_digital_inputs_I_172;
	::InputVariables[1,173] AT %IB."KUKA2_KRC4_ProfiNet_5_0".Module001_8_digital_inputs_I_173;
	::InputVariables[1,174] AT %IB."KUKA2_KRC4_ProfiNet_5_0".Module001_8_digital_inputs_I_174;
	::InputVariables[1,175] AT %IB."KUKA2_KRC4_ProfiNet_5_0".Module001_8_digital_inputs_I_175;
	::InputVariables[1,176] AT %IB."KUKA2_KRC4_ProfiNet_5_0".Module001_8_digital_inputs_I_176;
	::InputVariables[1,177] AT %IB."KUKA2_KRC4_ProfiNet_5_0".Module001_8_digital_inputs_I_177;
	::InputVariables[1,178] AT %IB."KUKA2_KRC4_ProfiNet_5_0".Module001_8_digital_inputs_I_178;
	::InputVariables[1,179] AT %IB."KUKA2_KRC4_ProfiNet_5_0".Module001_8_digital_inputs_I_179;
	::InputVariables[1,180] AT %IB."KUKA2_KRC4_ProfiNet_5_0".Module001_8_digital_inputs_I_180;
	::InputVariables[1,181] AT %IB."KUKA2_KRC4_ProfiNet_5_0".Module001_8_digital_inputs_I_181;
	::InputVariables[1,182] AT %IB."KUKA2_KRC4_ProfiNet_5_0".Module001_8_digital_inputs_I_182;
	::InputVariables[1,183] AT %IB."KUKA2_KRC4_ProfiNet_5_0".Module001_8_digital_inputs_I_183;
	::InputVariables[1,184] AT %IB."KUKA2_KRC4_ProfiNet_5_0".Module001_8_digital_inputs_I_184;
	::InputVariables[1,185] AT %IB."KUKA2_KRC4_ProfiNet_5_0".Module001_8_digital_inputs_I_185;
	::InputVariables[1,186] AT %IB."KUKA2_KRC4_ProfiNet_5_0".Module001_8_digital_inputs_I_186;
	::InputVariables[1,187] AT %IB."KUKA2_KRC4_ProfiNet_5_0".Module001_8_digital_inputs_I_187;
	::InputVariables[1,188] AT %IB."KUKA2_KRC4_ProfiNet_5_0".Module001_8_digital_inputs_I_188;
	::InputVariables[1,189] AT %IB."KUKA2_KRC4_ProfiNet_5_0".Module001_8_digital_inputs_I_189;
	::InputVariables[1,190] AT %IB."KUKA2_KRC4_ProfiNet_5_0".Module001_8_digital_inputs_I_190;
	::InputVariables[1,191] AT %IB."KUKA2_KRC4_ProfiNet_5_0".Module001_8_digital_inputs_I_191;
	::InputVariables[1,192] AT %IB."KUKA2_KRC4_ProfiNet_5_0".Module001_8_digital_inputs_I_192;
	::InputVariables[1,193] AT %IB."KUKA2_KRC4_ProfiNet_5_0".Module001_8_digital_inputs_I_193;
	::InputVariables[1,194] AT %IB."KUKA2_KRC4_ProfiNet_5_0".Module001_8_digital_inputs_I_194;
	::InputVariables[1,195] AT %IB."KUKA2_KRC4_ProfiNet_5_0".Module001_8_digital_inputs_I_195;
	::InputVariables[1,196] AT %IB."KUKA2_KRC4_ProfiNet_5_0".Module001_8_digital_inputs_I_196;
	::InputVariables[1,197] AT %IB."KUKA2_KRC4_ProfiNet_5_0".Module001_8_digital_inputs_I_197;
	::InputVariables[1,198] AT %IB."KUKA2_KRC4_ProfiNet_5_0".Module001_8_digital_inputs_I_198;
	::InputVariables[1,199] AT %IB."KUKA2_KRC4_ProfiNet_5_0".Module001_8_digital_inputs_I_199;
	::InputVariables[1,200] AT %IB."KUKA2_KRC4_ProfiNet_5_0".Module001_8_digital_inputs_I_200;
	::InputVariables[1,201] AT %IB."KUKA2_KRC4_ProfiNet_5_0".Module001_8_digital_inputs_I_201;
	::InputVariables[1,202] AT %IB."KUKA2_KRC4_ProfiNet_5_0".Module001_8_digital_inputs_I_202;
	::InputVariables[1,203] AT %IB."KUKA2_KRC4_ProfiNet_5_0".Module001_8_digital_inputs_I_203;
	::InputVariables[1,204] AT %IB."KUKA2_KRC4_ProfiNet_5_0".Module001_8_digital_inputs_I_204;
	::InputVariables[1,205] AT %IB."KUKA2_KRC4_ProfiNet_5_0".Module001_8_digital_inputs_I_205;
	::InputVariables[1,206] AT %IB."KUKA2_KRC4_ProfiNet_5_0".Module001_8_digital_inputs_I_206;
	::InputVariables[1,207] AT %IB."KUKA2_KRC4_ProfiNet_5_0".Module001_8_digital_inputs_I_207;
	::InputVariables[1,208] AT %IB."KUKA2_KRC4_ProfiNet_5_0".Module001_8_digital_inputs_I_208;
	::InputVariables[1,209] AT %IB."KUKA2_KRC4_ProfiNet_5_0".Module001_8_digital_inputs_I_209;
	::InputVariables[1,210] AT %IB."KUKA2_KRC4_ProfiNet_5_0".Module001_8_digital_inputs_I_210;
	::InputVariables[1,211] AT %IB."KUKA2_KRC4_ProfiNet_5_0".Module001_8_digital_inputs_I_211;
	::InputVariables[1,212] AT %IB."KUKA2_KRC4_ProfiNet_5_0".Module001_8_digital_inputs_I_212;
	::InputVariables[1,213] AT %IB."KUKA2_KRC4_ProfiNet_5_0".Module001_8_digital_inputs_I_213;
	::InputVariables[1,214] AT %IB."KUKA2_KRC4_ProfiNet_5_0".Module001_8_digital_inputs_I_214;
	::InputVariables[1,215] AT %IB."KUKA2_KRC4_ProfiNet_5_0".Module001_8_digital_inputs_I_215;
	::InputVariables[1,216] AT %IB."KUKA2_KRC4_ProfiNet_5_0".Module001_8_digital_inputs_I_216;
	::InputVariables[1,217] AT %IB."KUKA2_KRC4_ProfiNet_5_0".Module001_8_digital_inputs_I_217;
	::InputVariables[1,218] AT %IB."KUKA2_KRC4_ProfiNet_5_0".Module001_8_digital_inputs_I_218;
	::InputVariables[1,219] AT %IB."KUKA2_KRC4_ProfiNet_5_0".Module001_8_digital_inputs_I_219;
	::InputVariables[1,220] AT %IB."KUKA2_KRC4_ProfiNet_5_0".Module001_8_digital_inputs_I_220;
	::InputVariables[1,221] AT %IB."KUKA2_KRC4_ProfiNet_5_0".Module001_8_digital_inputs_I_221;
	::InputVariables[1,222] AT %IB."KUKA2_KRC4_ProfiNet_5_0".Module001_8_digital_inputs_I_222;
	::InputVariables[1,223] AT %IB."KUKA2_KRC4_ProfiNet_5_0".Module001_8_digital_inputs_I_223;
	::InputVariables[1,224] AT %IB."KUKA2_KRC4_ProfiNet_5_0".Module001_8_digital_inputs_I_224;
	::InputVariables[1,225] AT %IB."KUKA2_KRC4_ProfiNet_5_0".Module001_8_digital_inputs_I_225;
	::InputVariables[1,226] AT %IB."KUKA2_KRC4_ProfiNet_5_0".Module001_8_digital_inputs_I_226;
	::InputVariables[1,227] AT %IB."KUKA2_KRC4_ProfiNet_5_0".Module001_8_digital_inputs_I_227;
	::InputVariables[1,228] AT %IB."KUKA2_KRC4_ProfiNet_5_0".Module001_8_digital_inputs_I_228;
	::InputVariables[1,229] AT %IB."KUKA2_KRC4_ProfiNet_5_0".Module001_8_digital_inputs_I_229;
	::InputVariables[1,230] AT %IB."KUKA2_KRC4_ProfiNet_5_0".Module001_8_digital_inputs_I_230;
	::InputVariables[1,231] AT %IB."KUKA2_KRC4_ProfiNet_5_0".Module001_8_digital_inputs_I_231;
	::InputVariables[1,232] AT %IB."KUKA2_KRC4_ProfiNet_5_0".Module001_8_digital_inputs_I_232;
	::InputVariables[1,233] AT %IB."KUKA2_KRC4_ProfiNet_5_0".Module001_8_digital_inputs_I_233;
	::InputVariables[1,234] AT %IB."KUKA2_KRC4_ProfiNet_5_0".Module001_8_digital_inputs_I_234;
	::InputVariables[1,235] AT %IB."KUKA2_KRC4_ProfiNet_5_0".Module001_8_digital_inputs_I_235;
	::InputVariables[1,236] AT %IB."KUKA2_KRC4_ProfiNet_5_0".Module001_8_digital_inputs_I_236;
	::InputVariables[1,237] AT %IB."KUKA2_KRC4_ProfiNet_5_0".Module001_8_digital_inputs_I_237;
	::InputVariables[1,238] AT %IB."KUKA2_KRC4_ProfiNet_5_0".Module001_8_digital_inputs_I_238;
	::InputVariables[1,239] AT %IB."KUKA2_KRC4_ProfiNet_5_0".Module001_8_digital_inputs_I_239;
	::InputVariables[1,240] AT %IB."KUKA2_KRC4_ProfiNet_5_0".Module001_8_digital_inputs_I_240;
	::InputVariables[1,241] AT %IB."KUKA2_KRC4_ProfiNet_5_0".Module001_8_digital_inputs_I_241;
	::InputVariables[1,242] AT %IB."KUKA2_KRC4_ProfiNet_5_0".Module001_8_digital_inputs_I_242;
	::InputVariables[1,243] AT %IB."KUKA2_KRC4_ProfiNet_5_0".Module001_8_digital_inputs_I_243;
	::InputVariables[1,244] AT %IB."KUKA2_KRC4_ProfiNet_5_0".Module001_8_digital_inputs_I_244;
	::InputVariables[1,245] AT %IB."KUKA2_KRC4_ProfiNet_5_0".Module001_8_digital_inputs_I_245;
	::InputVariables[1,246] AT %IB."KUKA2_KRC4_ProfiNet_5_0".Module001_8_digital_inputs_I_246;
	::InputVariables[1,247] AT %IB."KUKA2_KRC4_ProfiNet_5_0".Module001_8_digital_inputs_I_247;
	::InputVariables[1,248] AT %IB."KUKA2_KRC4_ProfiNet_5_0".Module001_8_digital_inputs_I_248;
	::InputVariables[1,249] AT %IB."KUKA2_KRC4_ProfiNet_5_0".Module001_8_digital_inputs_I_249;
	::InputVariables[1,250] AT %IB."KUKA2_KRC4_ProfiNet_5_0".Module001_8_digital_inputs_I_250;
	::InputVariables[1,251] AT %IB."KUKA2_KRC4_ProfiNet_5_0".Module001_8_digital_inputs_I_251;
	::InputVariables[1,252] AT %IB."KUKA2_KRC4_ProfiNet_5_0".Module001_8_digital_inputs_I_252;
	::InputVariables[1,253] AT %IB."KUKA2_KRC4_ProfiNet_5_0".Module001_8_digital_inputs_I_253;
```
